KUKA KRL program: EPS_2_25990_SANMH03_A_20260122125456.src

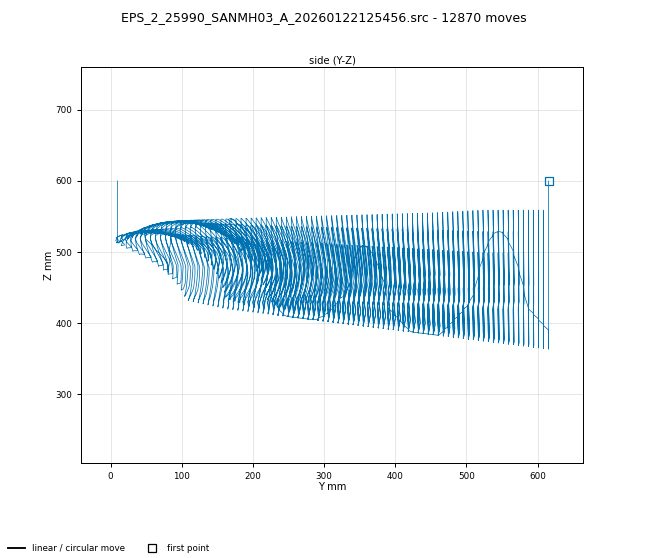
[picture p0: tool path of EPS_2_25990_SANMH03_A_20260122125456.src, 12870 of 12872 moves have a stored position in this frame; points joined in program order, loops and branches not executed]
&ACCESS RVP
&REL 4
&COMMENT QRS 19112012
&PARAM EDITMASK = *
DEF PART()
EXT BAS (BAS_COMMAND :IN,REAL :IN )
INT I
BAS (#INITMOV,0 )

;KUKA QRS Post kuka4.cps  Date:22-06-2017 !

File_ID=3006

QRS_PRE_INIT()

;Init var - Until changes are made in qrs_pre_init
Outlet_Square_prg=0
Inlet_1_Square_prg=0
Inlet_2_Square_prg=0
Inlet_3_Square_prg=0
Inlet_4_Square_prg=0
Inlet_5_Square_prg=0

Outlet_1={X 0.000, Y 520.860, Z 458.500, B 0.000, E1 0.000 }
Inlet_1={X 0.000, Y 523.030, Z 428.500, B 0.000, E1 121.000 }
Inlet_2={X 0.000, Y 529.760, Z 424.000, B 0.000, E1 213.000 }
Outlet_1_type=201
Inlet_1_type=201
Inlet_2_type=150
;QRS#1=Sidecore dimensions
;QRS#2=200-8" PVC SDR 35
;QRS#3=200-8" PVC SDR 35
;QRS#4=150-6" PVC SDR 28
;QRS#5=
;QRS#6=
;QRS#7=
;QRS#8=
;QRS#9=12-08 PSX
;QRS#10=12-08 PSX
;QRS#11=10-06 PSX
;QRS#12=
;QRS#13=
;QRS#14=
;QRS#15=
;QRS#16=1220x127x838 2,75'
;QRS#17=EPS Height
;QRS#18=559
;QRS#19=*
;QRS#20= UPDATED VERSION 22-06-2017
;QRS#21=*
Outlet_Square=0100
Inlet_1_Square=0100
Inlet_2_Square=070
Inlet_3_Square=0
Inlet_4_Square=0
Inlet_5_Square=0
Mill_Square=1
Outlet_Square_Prg=204
Inlet_1_Square_prg=204
Inlet_2_Square_prg=203

QRS_INIT()

$ADVANCE=5

; T1
PTP {E1 173.659,E2 173.659}
PTP {X 0,Y 615.494,A -85,B 0,C 180,E1 173.659,E2 173.659,E3 0,E4 0,E5 0,E6 0}
QRS_SPEED_INIT()
LIN {X 0,Y 615.494,Z 600,A -85,B 0,C 180,E1 173.659,E2 173.659,E3 0,E4 0,E5 0,E6 0} C_VEL
LIN {X 0,Y 615.494,Z 399.527,A -85,B 0,C 180,E1 173.659,E2 173.659} C_VEL
LIN {X 0,Y 615.494,Z 391.592,A -85,B 0,C 180,E1 173.659,E2 173.659} C_VEL
LIN {X 0,Y 615.477,Z 389.645,A -85,B 0,C 180,E1 173.431,E2 173.431} C_VEL
LIN {X 0,Y 615.481,Z 396.286,A -85,B 0,C 180,E1 170.801,E2 170.801} C_VEL
LIN {X 0,Y 615.485,Z 403.113,A -85,B 0,C 180,E1 168.139,E2 168.139} C_VEL
LIN {X 0,Y 615.478,Z 410.131,A -85,B 0,C 180,E1 165.451,E2 165.451} C_VEL
LIN {X 0,Y 615.485,Z 417.333,A -85,B 0,C 180,E1 162.73,E2 162.73} C_VEL
LIN {X 0,Y 615.493,Z 423.081,A -85,B 0,C 180,E1 160.576,E2 160.576} C_VEL
LIN {X 0,Y 615.483,Z 435.817,A -85,B 0,C 180,E1 160.315,E2 160.315} C_VEL
LIN {X 0,Y 615.464,Z 449.029,A -85,B 0,C 180,E1 159.902,E2 159.902} C_VEL
LIN {X 0,Y 615.483,Z 461.622,A -85,B 0,C 180,E1 159.358,E2 159.358} C_VEL
LIN {X 0,Y 615.489,Z 472.571,A -85,B 0,C 180,E1 158.744,E2 158.744} C_VEL
LIN {X 0,Y 615.498,Z 483.738,A -85,B 0,C 180,E1 157.952,E2 157.952} C_VEL
LIN {X 0,Y 615.498,Z 492.862,A -85,B 0,C 180,E1 157.156,E2 157.156} C_VEL
LIN {X 0,Y 615.497,Z 501.581,A -85,B 0,C 180,E1 156.217,E2 156.217} C_VEL
LIN {X 0,Y 615.498,Z 509.269,A -85,B 0,C 180,E1 155.189,E2 155.189} C_VEL
LIN {X 0,Y 615.498,Z 514.717,A -85,B 0,C 180,E1 154.285,E2 154.285} C_VEL
LIN {X 0,Y 615.499,Z 519.658,A -85,B 0,C 180,E1 153.256,E2 153.256} C_VEL
LIN {X 0,Y 615.496,Z 523.851,A -85,B 0,C 180,E1 152.086,E2 152.086} C_VEL
LIN {X 0,Y 615.495,Z 525.744,A -85,B 0,C 180,E1 151.343,E2 151.343} C_VEL
LIN {X 0,Y 615.499,Z 527.649,A -85,B 0,C 180,E1 150.204,E2 150.204} C_VEL
LIN {X 0,Y 615.492,Z 528.385,A -85,B 0,C 180,E1 148.914,E2 148.914} C_VEL
LIN {X 0,Y 615.497,Z 527.605,A -85,B 0,C 180,E1 147.668,E2 147.668} C_VEL
LIN {X 0,Y 615.497,Z 525.522,A -85,B 0,C 180,E1 146.465,E2 146.465} C_VEL
LIN {X 0,Y 615.499,Z 521.736,A -85,B 0,C 180,E1 145.186,E2 145.186} C_VEL
LIN {X 0,Y 615.497,Z 517.474,A -85,B 0,C 180,E1 144.166,E2 144.166} C_VEL
LIN {X 0,Y 615.497,Z 511.462,A -85,B 0,C 180,E1 143.063,E2 143.063} C_VEL
LIN {X 0,Y 615.494,Z 503.996,A -85,B 0,C 180,E1 141.988,E2 141.988} C_VEL
LIN {X 0,Y 615.498,Z 496.26,A -85,B 0,C 180,E1 141.097,E2 141.097} C_VEL
LIN {X 0,Y 615.495,Z 487.302,A -85,B 0,C 180,E1 140.251,E2 140.251} C_VEL
LIN {X 0,Y 615.498,Z 477.935,A -85,B 0,C 180,E1 139.524,E2 139.524} C_VEL
LIN {X 0,Y 615.427,Z 466.634,A -85,B 0,C 180,E1 138.814,E2 138.814} C_VEL
LIN {X 0,Y 615.417,Z 454.465,A -85,B 0,C 180,E1 138.223,E2 138.223} C_VEL
LIN {X 0,Y 615.453,Z 442.53,A -85,B 0,C 180,E1 137.786,E2 137.786} C_VEL
LIN {X 0,Y 615.497,Z 429.773,A -85,B 0,C 180,E1 137.457,E2 137.457} C_VEL
LIN {X 0,Y 615.475,Z 423.066,A -85,B 0,C 180,E1 137.327,E2 137.327} C_VEL
LIN {X 0,Y 615.428,Z 416.675,A -85,B 0,C 180,E1 134.926,E2 134.926} C_VEL
LIN {X 0,Y 615.42,Z 409.882,A -85,B 0,C 180,E1 132.359,E2 132.359} C_VEL
LIN {X 0,Y 615.486,Z 403.062,A -85,B 0,C 180,E1 129.751,E2 129.751} C_VEL
LIN {X 0,Y 615.43,Z 395.839,A -85,B 0,C 180,E1 126.93,E2 126.93} C_VEL
LIN {X 0,Y 615.426,Z 390.192,A -85,B 0,C 180,E1 124.693,E2 124.693} C_VEL
LIN {X 0,Y 615.446,Z 384.318,A -85,B 0,C 180,E1 122.325,E2 122.325} C_VEL
LIN {X 0,Y 615.466,Z 377.257,A -85,B 0,C 180,E1 119.408,E2 119.408} C_VEL
LIN {X 0,Y 615.473,Z 371.567,A -85,B 0,C 180,E1 117.043,E2 117.043} C_VEL
LIN {X 0,Y 615.487,Z 364.488,A -85,B 0,C 180,E1 114.273,E2 114.273} C_VEL
LIN {X 0,Y 615.495,Z 363.693,A -85,B 0,C 180,E1 113.897,E2 113.897} C_VEL
LIN {X 0,Y 615.487,Z 363.694,A -85,B 0,C 180,E1 111.433,E2 111.433} C_VEL
LIN {X 0,Y 615.445,Z 363.7,A -85,B 0,C 180,E1 108.594,E2 108.594} C_VEL
LIN {X 0,Y 615.49,Z 363.691,A -85,B 0,C 180,E1 105.906,E2 105.906} C_VEL
LIN {X 0,Y 615.492,Z 363.7,A -85,B 0,C 180,E1 103.202,E2 103.202} C_VEL
LIN {X 0,Y 615.458,Z 363.7,A -85,B 0,C 180,E1 100.529,E2 100.529} C_VEL
LIN {X 0,Y 615.489,Z 363.69,A -85,B 0,C 180,E1 97.877,E2 97.877} C_VEL
LIN {X 0,Y 615.476,Z 363.7,A -85,B 0,C 180,E1 95.243,E2 95.243} C_VEL
LIN {X 0,Y 615.461,Z 363.701,A -85,B 0,C 180,E1 92.619,E2 92.619} C_VEL
LIN {X 0,Y 615.485,Z 363.692,A -85,B 0,C 180,E1 89.674,E2 89.674} C_VEL
LIN {X 0,Y 615.49,Z 363.848,A -85,B 0,C 180,E1 89.347,E2 89.347} C_VEL
LIN {X 0,Y 615.489,Z 369.621,A -85,B 0,C 180,E1 86.729,E2 86.729} C_VEL
LIN {X 0,Y 615.496,Z 375.508,A -85,B 0,C 180,E1 84.103,E2 84.103} C_VEL
LIN {X 0,Y 615.474,Z 381.581,A -85,B 0,C 180,E1 81.465,E2 81.465} C_VEL
LIN {X 0,Y 615.479,Z 387.798,A -85,B 0,C 180,E1 78.809,E2 78.809} C_VEL
LIN {X 0,Y 615.494,Z 394.357,A -85,B 0,C 180,E1 76.064,E2 76.064} C_VEL
LIN {X 0,Y 615.485,Z 400.781,A -85,B 0,C 180,E1 73.415,E2 73.415} C_VEL
LIN {X 0,Y 615.459,Z 407.558,A -85,B 0,C 180,E1 70.663,E2 70.663} C_VEL
LIN {X 0,Y 615.493,Z 414.508,A -85,B 0,C 180,E1 67.866,E2 67.866} C_VEL
LIN {X 0,Y 615.496,Z 419.067,A -85,B 0,C 180,E1 66.103,E2 66.103} C_VEL
LIN {X 0,Y 615.478,Z 430.982,A -85,B 0,C 180,E1 65.794,E2 65.794} C_VEL
LIN {X 0,Y 615.446,Z 439.974,A -85,B 0,C 180,E1 65.459,E2 65.459} C_VEL
LIN {X 0,Y 615.436,Z 449.191,A -85,B 0,C 180,E1 65.008,E2 65.008} C_VEL
LIN {X 0,Y 615.47,Z 457.359,A -85,B 0,C 180,E1 64.504,E2 64.504} C_VEL
LIN {X 0,Y 615.499,Z 465.031,A -85,B 0,C 180,E1 63.923,E2 63.923} C_VEL
LIN {X 0,Y 615.496,Z 473.758,A -85,B 0,C 180,E1 63.104,E2 63.104} C_VEL
LIN {X 0,Y 615.499,Z 480.59,A -85,B 0,C 180,E1 62.273,E2 62.273} C_VEL
LIN {X 0,Y 615.497,Z 485.434,A -85,B 0,C 180,E1 61.548,E2 61.548} C_VEL
LIN {X 0,Y 615.492,Z 488.696,A -85,B 0,C 180,E1 60.971,E2 60.971} C_VEL
LIN {X 0,Y 615.498,Z 492.162,A -85,B 0,C 180,E1 60.203,E2 60.203} C_VEL
LIN {X 0,Y 615.496,Z 494.722,A -85,B 0,C 180,E1 59.464,E2 59.464} C_VEL
LIN {X 0,Y 615.495,Z 497.253,A -85,B 0,C 180,E1 58.318,E2 58.318} C_VEL
LIN {X 0,Y 615.496,Z 498.133,A -85,B 0,C 180,E1 57.546,E2 57.546} C_VEL
LIN {X 0,Y 615.492,Z 498.18,A -85,B 0,C 180,E1 56.465,E2 56.465} C_VEL
LIN {X 0,Y 615.492,Z 496.809,A -85,B 0,C 180,E1 55.298,E2 55.298} C_VEL
LIN {X 0,Y 615.491,Z 493.761,A -85,B 0,C 180,E1 54.166,E2 54.166} C_VEL
LIN {X 0,Y 615.497,Z 490.45,A -85,B 0,C 180,E1 53.321,E2 53.321} C_VEL
LIN {X 0,Y 615.493,Z 486.628,A -85,B 0,C 180,E1 52.568,E2 52.568} C_VEL
LIN {X 0,Y 615.496,Z 482.71,A -85,B 0,C 180,E1 51.935,E2 51.935} C_VEL
LIN {X 0,Y 615.498,Z 476.29,A -85,B 0,C 180,E1 51.099,E2 51.099} C_VEL
LIN {X 0,Y 615.499,Z 469.919,A -85,B 0,C 180,E1 50.425,E2 50.425} C_VEL
LIN {X 0,Y 615.474,Z 460.924,A -85,B 0,C 180,E1 49.652,E2 49.652} C_VEL
LIN {X 0,Y 615.455,Z 451.474,A -85,B 0,C 180,E1 49.03,E2 49.03} C_VEL
LIN {X 0,Y 615.487,Z 442.766,A -85,B 0,C 180,E1 48.577,E2 48.577} C_VEL
LIN {X 0,Y 615.494,Z 434.152,A -85,B 0,C 180,E1 48.225,E2 48.225} C_VEL
LIN {X 0,Y 615.491,Z 425.461,A -85,B 0,C 180,E1 47.958,E2 47.958} C_VEL
LIN {X 0,Y 615.48,Z 418.875,A -85,B 0,C 180,E1 47.784,E2 47.784} C_VEL
LIN {X 0,Y 615.455,Z 411.74,A -85,B 0,C 180,E1 44.932,E2 44.932} C_VEL
LIN {X 0,Y 615.469,Z 404.683,A -85,B 0,C 180,E1 42.082,E2 42.082} C_VEL
LIN {X 0,Y 615.426,Z 398.996,A -85,B 0,C 180,E1 39.755,E2 39.755} C_VEL
LIN {X 0,Y 615.43,Z 394.77,A -85,B 0,C 180,E1 38.009,E2 38.009} C_VEL
LIN {X 0,Y 615.423,Z 389.043,A -85,B 0,C 180,E1 35.62,E2 35.62} C_VEL
LIN {X 0,Y 615.455,Z 383.422,A -85,B 0,C 180,E1 33.238,E2 33.238} C_VEL
LIN {X 0,Y 615.491,Z 378.051,A -85,B 0,C 180,E1 30.919,E2 30.919} C_VEL
LIN {X 0,Y 615.473,Z 372.464,A -85,B 0,C 180,E1 28.453,E2 28.453} C_VEL
LIN {X 0,Y 615.494,Z 366.375,A -85,B 0,C 180,E1 25.715,E2 25.715} C_VEL
LIN {X 0,Y 615.473,Z 363.7,A -85,B 0,C 180,E1 24.452,E2 24.452} C_VEL
LIN {X 0,Y 615.496,Z 363.699,A -85,B 0,C 180,E1 22.136,E2 22.136} C_VEL
LIN {X 0,Y 615.489,Z 363.701,A -85,B 0,C 180,E1 19.338,E2 19.338} C_VEL
LIN {X 0,Y 615.485,Z 363.7,A -85,B 0,C 180,E1 16.586,E2 16.586} C_VEL
LIN {X 0,Y 615.483,Z 363.699,A -85,B 0,C 180,E1 13.874,E2 13.874} C_VEL
LIN {X 0,Y 615.489,Z 363.694,A -85,B 0,C 180,E1 10.904,E2 10.904} C_VEL
LIN {X 0,Y 615.482,Z 363.7,A -85,B 0,C 180,E1 8.536,E2 8.536} C_VEL
LIN {X 0,Y 615.487,Z 363.7,A -85,B 0,C 180,E1 5.898,E2 5.898} C_VEL
LIN {X 0,Y 615.492,Z 363.7,A -85,B 0,C 180,E1 3.273,E2 3.273} C_VEL
LIN {X 0,Y 615.489,Z 363.701,A -85,B 0,C 180,E1 0.654,E2 0.654} C_VEL
LIN {X 0,Y 615.498,Z 363.7,A -85,B 0,C 180,E1 -1.963,E2 -1.963} C_VEL
LIN {X 0,Y 615.489,Z 363.701,A -85,B 0,C 180,E1 -4.585,E2 -4.585} C_VEL
LIN {X 0,Y 615.492,Z 363.699,A -85,B 0,C 180,E1 -7.216,E2 -7.216} C_VEL
LIN {X 0,Y 615.487,Z 363.7,A -85,B 0,C 180,E1 -9.862,E2 -9.862} C_VEL
LIN {X 0,Y 615.485,Z 363.7,A -85,B 0,C 180,E1 -12.53,E2 -12.53} C_VEL
LIN {X 0,Y 615.491,Z 363.699,A -85,B 0,C 180,E1 -15.226,E2 -15.226} C_VEL
LIN {X 0,Y 615.49,Z 363.701,A -85,B 0,C 180,E1 -17.957,E2 -17.957} C_VEL
LIN {X 0,Y 615.492,Z 363.701,A -85,B 0,C 180,E1 -20.731,E2 -20.731} C_VEL
LIN {X 0,Y 615.478,Z 363.7,A -85,B 0,C 180,E1 -23.557,E2 -23.557} C_VEL
LIN {X 0,Y 615.488,Z 363.695,A -85,B 0,C 180,E1 -26.444,E2 -26.444} C_VEL
LIN {X 0,Y 615.459,Z 363.7,A -85,B 0,C 180,E1 -29.408,E2 -29.408} C_VEL
LIN {X 0,Y 615.472,Z 363.7,A -85,B 0,C 180,E1 -31.687,E2 -31.687} C_VEL
LIN {X 0,Y 615.492,Z 363.692,A -85,B 0,C 180,E1 -34.706,E2 -34.706} C_VEL
LIN {X 0,Y 615.457,Z 363.701,A -85,B 0,C 180,E1 -37.245,E2 -37.245} C_VEL
LIN {X 0,Y 615.473,Z 363.699,A -85,B 0,C 180,E1 -39.752,E2 -39.752} C_VEL
LIN {X 0,Y 615.495,Z 363.695,A -85,B 0,C 180,E1 -42.353,E2 -42.353} C_VEL
LIN {X 0,Y 615.468,Z 363.7,A -85,B 0,C 180,E1 -45.071,E2 -45.071} C_VEL
LIN {X 0,Y 615.474,Z 363.697,A -85,B 0,C 180,E1 -47.922,E2 -47.922} C_VEL
LIN {X 0,Y 615.477,Z 363.697,A -85,B 0,C 180,E1 -50.94,E2 -50.94} C_VEL
LIN {X 0,Y 615.46,Z 363.7,A -85,B 0,C 180,E1 -53.576,E2 -53.576} C_VEL
LIN {X 0,Y 615.492,Z 363.695,A -85,B 0,C 180,E1 -56.466,E2 -56.466} C_VEL
LIN {X 0,Y 615.477,Z 363.698,A -85,B 0,C 180,E1 -59.082,E2 -59.082} C_VEL
LIN {X 0,Y 615.49,Z 363.711,A -85,B 0,C 180,E1 -60.303,E2 -60.303} C_VEL
LIN {X 0,Y 615.449,Z 375.744,A -85,B 0,C 180,E1 -62.963,E2 -62.963} C_VEL
LIN {X 0,Y 615.43,Z 385.189,A -85,B 0,C 180,E1 -65.008,E2 -65.008} C_VEL
LIN {X 0,Y 615.446,Z 396.451,A -85,B 0,C 180,E1 -67.408,E2 -67.408} C_VEL
LIN {X 0,Y 615.494,Z 408.677,A -85,B 0,C 180,E1 -69.97,E2 -69.97} C_VEL
LIN {X 0,Y 615.472,Z 422.09,A -85,B 0,C 180,E1 -72.731,E2 -72.731} C_VEL
LIN {X 0,Y 615.475,Z 435.487,A -85,B 0,C 180,E1 -75.453,E2 -75.453} C_VEL
LIN {X 0,Y 615.488,Z 448.873,A -85,B 0,C 180,E1 -78.141,E2 -78.141} C_VEL
LIN {X 0,Y 615.494,Z 449.811,A -85,B 0,C 180,E1 -78.329,E2 -78.329} C_VEL
LIN {X 0,Y 615.498,Z 464.14,A -85,B 0,C 180,E1 -78.6,E2 -78.6} C_VEL
LIN {X 0,Y 615.463,Z 476.758,A -85,B 0,C 180,E1 -78.969,E2 -78.969} C_VEL
LIN {X 0,Y 615.451,Z 489.065,A -85,B 0,C 180,E1 -79.474,E2 -79.474} C_VEL
LIN {X 0,Y 615.486,Z 500.011,A -85,B 0,C 180,E1 -80.057,E2 -80.057} C_VEL
LIN {X 0,Y 615.499,Z 511.19,A -85,B 0,C 180,E1 -80.803,E2 -80.803} C_VEL
LIN {X 0,Y 615.498,Z 521.063,A -85,B 0,C 180,E1 -81.631,E2 -81.631} C_VEL
LIN {X 0,Y 615.498,Z 530.62,A -85,B 0,C 180,E1 -82.621,E2 -82.621} C_VEL
LIN {X 0,Y 615.496,Z 538.214,A -85,B 0,C 180,E1 -83.61,E2 -83.61} C_VEL
LIN {X 0,Y 615.498,Z 545.213,A -85,B 0,C 180,E1 -84.76,E2 -84.76} C_VEL
LIN {X 0,Y 615.494,Z 549.858,A -85,B 0,C 180,E1 -85.745,E2 -85.745} C_VEL
LIN {X 0,Y 615.494,Z 553.404,A -85,B 0,C 180,E1 -86.729,E2 -86.729} C_VEL
LIN {X 0,Y 615.497,Z 555.237,A -85,B 0,C 180,E1 -87.384,E2 -87.384} C_VEL
LIN {X 0,Y 615.499,Z 556.61,A -85,B 0,C 180,E1 -88.038,E2 -88.038} C_VEL
LIN {X 0,Y 615.496,Z 558.175,A -85,B 0,C 180,E1 -89.347,E2 -89.347} C_VEL
LIN {X 0,Y 615.494,Z 558.389,A -85,B 0,C 180,E1 -90.001,E2 -90.001} C_VEL
LIN {X 0,Y 615.495,Z 557.578,A -85,B 0,C 180,E1 -91.31,E2 -91.31} C_VEL
LIN {X 0,Y 615.499,Z 556.605,A -85,B 0,C 180,E1 -91.964,E2 -91.964} C_VEL
LIN {X 0,Y 615.497,Z 555.229,A -85,B 0,C 180,E1 -92.619,E2 -92.619} C_VEL
LIN {X 0,Y 615.496,Z 552.345,A -85,B 0,C 180,E1 -93.602,E2 -93.602} C_VEL
LIN {X 0,Y 615.498,Z 548.436,A -85,B 0,C 180,E1 -94.586,E2 -94.586} C_VEL
LIN {X 0,Y 615.499,Z 543.397,A -85,B 0,C 180,E1 -95.571,E2 -95.571} C_VEL
LIN {X 0,Y 615.497,Z 536.87,A -85,B 0,C 180,E1 -96.583,E2 -96.583} C_VEL
LIN {X 0,Y 615.497,Z 529.122,A -85,B 0,C 180,E1 -97.547,E2 -97.547} C_VEL
LIN {X 0,Y 615.498,Z 521.031,A -85,B 0,C 180,E1 -98.372,E2 -98.372} C_VEL
LIN {X 0,Y 615.499,Z 511.151,A -85,B 0,C 180,E1 -99.2,E2 -99.2} C_VEL
LIN {X 0,Y 615.488,Z 499.961,A -85,B 0,C 180,E1 -99.946,E2 -99.946} C_VEL
LIN {X 0,Y 615.452,Z 489.003,A -85,B 0,C 180,E1 -100.529,E2 -100.529} C_VEL
LIN {X 0,Y 615.464,Z 476.705,A -85,B 0,C 180,E1 -101.033,E2 -101.033} C_VEL
LIN {X 0,Y 615.498,Z 464.01,A -85,B 0,C 180,E1 -101.403,E2 -101.403} C_VEL
LIN {X 0,Y 615.494,Z 449.797,A -85,B 0,C 180,E1 -101.674,E2 -101.674} C_VEL
LIN {X 0,Y 615.475,Z 437.007,A -85,B 0,C 180,E1 -104.242,E2 -104.242} C_VEL
LIN {X 0,Y 615.481,Z 423.747,A -85,B 0,C 180,E1 -106.93,E2 -106.93} C_VEL
LIN {X 0,Y 615.483,Z 410.342,A -85,B 0,C 180,E1 -109.686,E2 -109.686} C_VEL
LIN {X 0,Y 615.467,Z 397.638,A -85,B 0,C 180,E1 -112.341,E2 -112.341} C_VEL
LIN {X 0,Y 615.427,Z 386.854,A -85,B 0,C 180,E1 -114.635,E2 -114.635} C_VEL
LIN {X 0,Y 615.449,Z 375.744,A -85,B 0,C 180,E1 -117.037,E2 -117.037} C_VEL
LIN {X 0,Y 615.485,Z 363.69,A -85,B 0,C 180,E1 -119.721,E2 -119.721} C_VEL
LIN {X 0,Y 615.472,Z 363.695,A -85,B 0,C 180,E1 -122.459,E2 -122.459} C_VEL
LIN {X 0,Y 615.486,Z 363.697,A -85,B 0,C 180,E1 -124.816,E2 -124.816} C_VEL
LIN {X 0,Y 615.474,Z 363.689,A -85,B 0,C 180,E1 -127.244,E2 -127.244} C_VEL
LIN {X 0,Y 615.488,Z 363.7,A -85,B 0,C 180,E1 -130.089,E2 -130.089} C_VEL
LIN {X 0,Y 615.439,Z 363.699,A -85,B 0,C 180,E1 -132.358,E2 -132.358} C_VEL
LIN {X 0,Y 615.455,Z 363.701,A -85,B 0,C 180,E1 -135.072,E2 -135.072} C_VEL
LIN {X 0,Y 615.456,Z 363.693,A -85,B 0,C 180,E1 -137.924,E2 -137.924} C_VEL
LIN {X 0,Y 615.463,Z 363.695,A -85,B 0,C 180,E1 -140.248,E2 -140.248} C_VEL
LIN {X 0,Y 615.483,Z 363.69,A -85,B 0,C 180,E1 -143.064,E2 -143.064} C_VEL
LIN {X 0,Y 615.488,Z 363.686,A -85,B 0,C 180,E1 -145.3,E2 -145.3} C_VEL
LIN {X 0,Y 615.493,Z 363.694,A -85,B 0,C 180,E1 -147.669,E2 -147.669} C_VEL
LIN {X 0,Y 615.448,Z 363.698,A -85,B 0,C 180,E1 -150.212,E2 -150.212} C_VEL
LIN {X 0,Y 615.435,Z 363.7,A -85,B 0,C 180,E1 -152.082,E2 -152.082} C_VEL
LIN {X 0,Y 615.431,Z 363.7,A -85,B 0,C 180,E1 -154.443,E2 -154.443} C_VEL
LIN {X 0,Y 615.497,Z 363.692,A -85,B 0,C 180,E1 -157.156,E2 -157.156} C_VEL
LIN {X 0,Y 615.461,Z 363.695,A -85,B 0,C 180,E1 -159.966,E2 -159.966} C_VEL
LIN {X 0,Y 615.48,Z 363.691,A -85,B 0,C 180,E1 -162.729,E2 -162.729} C_VEL
LIN {X 0,Y 615.49,Z 363.691,A -85,B 0,C 180,E1 -165.451,E2 -165.451} C_VEL
LIN {X 0,Y 615.454,Z 363.697,A -85,B 0,C 180,E1 -168.138,E2 -168.138} C_VEL
LIN {X 0,Y 615.462,Z 363.697,A -85,B 0,C 180,E1 -170.801,E2 -170.801} C_VEL
LIN {X 0,Y 615.453,Z 363.698,A -85,B 0,C 180,E1 -173.45,E2 -173.45} C_VEL
LIN {X 0,Y 615.449,Z 363.698,A -85,B 0,C 180,E1 -176.071,E2 -176.071} C_VEL
LIN {X 0,Y 615.476,Z 363.974,A -85,B 0,C 180,E1 -176.399,E2 -176.399} C_VEL
LIN {X 0,Y 615.489,Z 370.297,A -85,B 0,C 180,E1 -178.691,E2 -178.691} C_VEL
LIN {X 0,Y 615.482,Z 375.236,A -85,B 0,C 180,E1 -180.654,E2 -180.654} C_VEL
LIN {X 0,Y 615.48,Z 381.527,A -85,B 0,C 180,E1 -183.273,E2 -183.273} C_VEL
LIN {X 0,Y 615.497,Z 387.971,A -85,B 0,C 180,E1 -185.898,E2 -185.898} C_VEL
LIN {X 0,Y 615.477,Z 389.645,A -85,B 0,C 180,E1 -186.569,E2 -186.569} C_VEL
LIN {X 0,Y 614.8,Z 391.13,A -85,B 0,C 180,E1 -187.099,E2 -187.099} C_VEL
LIN {X 0,Y 611.944,Z 393.686,A -85,B 0,C 180,E1 -187.953,E2 -187.953} C_VEL
LIN {X 0,Y 609.543,Z 395.676,A -85,B 0,C 180,E1 -188.64,E2 -188.64} C_VEL
LIN {X 0,Y 608.513,Z 397.105,A -85,B 0,C 180,E1 -189.172,E2 -189.172} C_VEL
LIN {X 0,Y 608.431,Z 397.568,A -85,B 0,C 180,E1 -189.353,E2 -189.353} C_VEL
LIN {X 0,Y 608.425,Z 404.335,A -85,B 0,C 180,E1 -192,E2 -192} C_VEL
LIN {X 0,Y 608.436,Z 411.401,A -85,B 0,C 180,E1 -194.721,E2 -194.721} C_VEL
LIN {X 0,Y 608.429,Z 418.66,A -85,B 0,C 180,E1 -197.477,E2 -197.477} C_VEL
LIN {X 0,Y 608.432,Z 423.472,A -85,B 0,C 180,E1 -199.286,E2 -199.286} C_VEL
LIN {X 0,Y 608.523,Z 438.048,A -85,B 0,C 180,E1 -199.612,E2 -199.612} C_VEL
LIN {X 0,Y 608.503,Z 451.304,A -85,B 0,C 180,E1 -200.052,E2 -200.052} C_VEL
LIN {X 0,Y 608.513,Z 463.064,A -85,B 0,C 180,E1 -200.587,E2 -200.587} C_VEL
LIN {X 0,Y 608.486,Z 474.347,A -85,B 0,C 180,E1 -201.246,E2 -201.246} C_VEL
LIN {X 0,Y 608.497,Z 485.298,A -85,B 0,C 180,E1 -202.047,E2 -202.047} C_VEL
LIN {X 0,Y 608.475,Z 494.924,A -85,B 0,C 180,E1 -202.925,E2 -202.925} C_VEL
LIN {X 0,Y 608.445,Z 503.147,A -85,B 0,C 180,E1 -203.846,E2 -203.846} C_VEL
LIN {X 0,Y 608.456,Z 510.996,A -85,B 0,C 180,E1 -204.935,E2 -204.935} C_VEL
LIN {X 0,Y 608.437,Z 517.174,A -85,B 0,C 180,E1 -206.036,E2 -206.036} C_VEL
LIN {X 0,Y 608.435,Z 522.153,A -85,B 0,C 180,E1 -207.199,E2 -207.199} C_VEL
LIN {X 0,Y 608.441,Z 525.464,A -85,B 0,C 180,E1 -208.267,E2 -208.267} C_VEL
LIN {X 0,Y 608.42,Z 527.14,A -85,B 0,C 180,E1 -209.022,E2 -209.022} C_VEL
LIN {X 0,Y 608.423,Z 528.469,A -85,B 0,C 180,E1 -209.964,E2 -209.964} C_VEL
LIN {X 0,Y 608.439,Z 528.887,A -85,B 0,C 180,E1 -210.546,E2 -210.546} C_VEL
LIN {X 0,Y 608.422,Z 528.942,A -85,B 0,C 180,E1 -211.319,E2 -211.319} C_VEL
LIN {X 0,Y 608.422,Z 528.01,A -85,B 0,C 180,E1 -212.516,E2 -212.516} C_VEL
LIN {X 0,Y 608.424,Z 525.719,A -85,B 0,C 180,E1 -213.727,E2 -213.727} C_VEL
LIN {X 0,Y 608.429,Z 522.112,A -85,B 0,C 180,E1 -214.902,E2 -214.902} C_VEL
LIN {X 0,Y 608.456,Z 516.993,A -85,B 0,C 180,E1 -216.091,E2 -216.091} C_VEL
LIN {X 0,Y 608.439,Z 511.004,A -85,B 0,C 180,E1 -217.154,E2 -217.154} C_VEL
LIN {X 0,Y 608.458,Z 503.196,A -85,B 0,C 180,E1 -218.238,E2 -218.238} C_VEL
LIN {X 0,Y 608.483,Z 495.025,A -85,B 0,C 180,E1 -219.155,E2 -219.155} C_VEL
LIN {X 0,Y 608.489,Z 486.121,A -85,B 0,C 180,E1 -219.976,E2 -219.976} C_VEL
LIN {X 0,Y 608.482,Z 476,A -85,B 0,C 180,E1 -220.736,E2 -220.736} C_VEL
LIN {X 0,Y 608.428,Z 464.384,A -85,B 0,C 180,E1 -221.434,E2 -221.434} C_VEL
LIN {X 0,Y 608.456,Z 452.111,A -85,B 0,C 180,E1 -222.007,E2 -222.007} C_VEL
LIN {X 0,Y 608.513,Z 439.113,A -85,B 0,C 180,E1 -222.449,E2 -222.449} C_VEL
LIN {X 0,Y 608.539,Z 425.565,A -85,B 0,C 180,E1 -222.757,E2 -222.757} C_VEL
LIN {X 0,Y 608.414,Z 423.473,A -85,B 0,C 180,E1 -222.804,E2 -222.804} C_VEL
LIN {X 0,Y 608.362,Z 417.125,A -85,B 0,C 180,E1 -225.195,E2 -225.195} C_VEL
LIN {X 0,Y 608.383,Z 409.935,A -85,B 0,C 180,E1 -227.931,E2 -227.931} C_VEL
LIN {X 0,Y 608.418,Z 402.744,A -85,B 0,C 180,E1 -230.708,E2 -230.708} C_VEL
LIN {X 0,Y 608.395,Z 395.662,A -85,B 0,C 180,E1 -233.493,E2 -233.493} C_VEL
LIN {X 0,Y 608.445,Z 388.591,A -85,B 0,C 180,E1 -236.327,E2 -236.327} C_VEL
LIN {X 0,Y 608.434,Z 382.719,A -85,B 0,C 180,E1 -238.734,E2 -238.734} C_VEL
LIN {X 0,Y 608.41,Z 377.366,A -85,B 0,C 180,E1 -240.976,E2 -240.976} C_VEL
LIN {X 0,Y 608.429,Z 371.805,A -85,B 0,C 180,E1 -243.224,E2 -243.224} C_VEL
LIN {X 0,Y 608.46,Z 365.141,A -85,B 0,C 180,E1 -245.851,E2 -245.851} C_VEL
LIN {X 0,Y 608.48,Z 364.69,A -85,B 0,C 180,E1 -246.155,E2 -246.155} C_VEL
LIN {X 0,Y 608.468,Z 364.69,A -85,B 0,C 180,E1 -248.307,E2 -248.307} C_VEL
LIN {X 0,Y 608.437,Z 364.693,A -85,B 0,C 180,E1 -251.129,E2 -251.129} C_VEL
LIN {X 0,Y 608.464,Z 364.693,A -85,B 0,C 180,E1 -253.905,E2 -253.905} C_VEL
LIN {X 0,Y 608.47,Z 364.695,A -85,B 0,C 180,E1 -256.643,E2 -256.643} C_VEL
LIN {X 0,Y 608.433,Z 364.695,A -85,B 0,C 180,E1 -259.348,E2 -259.348} C_VEL
LIN {X 0,Y 608.481,Z 364.688,A -85,B 0,C 180,E1 -262.032,E2 -262.032} C_VEL
LIN {X 0,Y 608.458,Z 364.696,A -85,B 0,C 180,E1 -264.697,E2 -264.697} C_VEL
LIN {X 0,Y 608.453,Z 364.694,A -85,B 0,C 180,E1 -267.35,E2 -267.35} C_VEL
LIN {X 0,Y 608.48,Z 364.688,A -85,B 0,C 180,E1 -269.999,E2 -269.999} C_VEL
LIN {X 0,Y 608.484,Z 364.881,A -85,B 0,C 180,E1 -270.66,E2 -270.66} C_VEL
LIN {X 0,Y 608.453,Z 370.695,A -85,B 0,C 180,E1 -273.309,E2 -273.309} C_VEL
LIN {X 0,Y 608.466,Z 376.611,A -85,B 0,C 180,E1 -275.965,E2 -275.965} C_VEL
LIN {X 0,Y 608.447,Z 382.709,A -85,B 0,C 180,E1 -278.634,E2 -278.634} C_VEL
LIN {X 0,Y 608.442,Z 388.979,A -85,B 0,C 180,E1 -281.323,E2 -281.323} C_VEL
LIN {X 0,Y 608.446,Z 395.428,A -85,B 0,C 180,E1 -284.036,E2 -284.036} C_VEL
LIN {X 0,Y 608.438,Z 402.064,A -85,B 0,C 180,E1 -286.783,E2 -286.783} C_VEL
LIN {X 0,Y 608.419,Z 407.168,A -85,B 0,C 180,E1 -288.869,E2 -288.869} C_VEL
LIN {X 0,Y 608.401,Z 414.149,A -85,B 0,C 180,E1 -291.692,E2 -291.692} C_VEL
LIN {X 0,Y 608.44,Z 419.345,A -85,B 0,C 180,E1 -293.776,E2 -293.776} C_VEL
LIN {X 0,Y 608.483,Z 431.922,A -85,B 0,C 180,E1 -294.124,E2 -294.124} C_VEL
LIN {X 0,Y 608.442,Z 440.087,A -85,B 0,C 180,E1 -294.434,E2 -294.434} C_VEL
LIN {X 0,Y 608.41,Z 448.545,A -85,B 0,C 180,E1 -294.844,E2 -294.844} C_VEL
LIN {X 0,Y 608.443,Z 457.188,A -85,B 0,C 180,E1 -295.372,E2 -295.372} C_VEL
LIN {X 0,Y 608.481,Z 465.852,A -85,B 0,C 180,E1 -296.032,E2 -296.032} C_VEL
LIN {X 0,Y 608.448,Z 473.694,A -85,B 0,C 180,E1 -296.772,E2 -296.772} C_VEL
LIN {X 0,Y 608.443,Z 481.324,A -85,B 0,C 180,E1 -297.703,E2 -297.703} C_VEL
LIN {X 0,Y 608.445,Z 486.166,A -85,B 0,C 180,E1 -298.438,E2 -298.438} C_VEL
LIN {X 0,Y 608.426,Z 489.398,A -85,B 0,C 180,E1 -299.02,E2 -299.02} C_VEL
LIN {X 0,Y 608.438,Z 493.447,A -85,B 0,C 180,E1 -299.967,E2 -299.967} C_VEL
LIN {X 0,Y 608.441,Z 495.409,A -85,B 0,C 180,E1 -300.544,E2 -300.544} C_VEL
LIN {X 0,Y 608.441,Z 497.293,A -85,B 0,C 180,E1 -301.315,E2 -301.315} C_VEL
LIN {X 0,Y 608.42,Z 498.463,A -85,B 0,C 180,E1 -302.095,E2 -302.095} C_VEL
LIN {X 0,Y 608.415,Z 498.947,A -85,B 0,C 180,E1 -302.879,E2 -302.879} C_VEL
LIN {X 0,Y 608.419,Z 498.704,A -85,B 0,C 180,E1 -303.728,E2 -303.728} C_VEL
LIN {X 0,Y 608.428,Z 496.988,A -85,B 0,C 180,E1 -304.903,E2 -304.903} C_VEL
LIN {X 0,Y 608.426,Z 494.97,A -85,B 0,C 180,E1 -305.682,E2 -305.682} C_VEL
LIN {X 0,Y 608.452,Z 492.006,A -85,B 0,C 180,E1 -306.5,E2 -306.5} C_VEL
LIN {X 0,Y 608.428,Z 487.485,A -85,B 0,C 180,E1 -307.423,E2 -307.423} C_VEL
LIN {X 0,Y 608.455,Z 482.373,A -85,B 0,C 180,E1 -308.239,E2 -308.239} C_VEL
LIN {X 0,Y 608.464,Z 476.379,A -85,B 0,C 180,E1 -309.01,E2 -309.01} C_VEL
LIN {X 0,Y 608.467,Z 469.222,A -85,B 0,C 180,E1 -309.759,E2 -309.759} C_VEL
LIN {X 0,Y 608.449,Z 460.418,A -85,B 0,C 180,E1 -310.496,E2 -310.496} C_VEL
LIN {X 0,Y 608.451,Z 451.779,A -85,B 0,C 180,E1 -311.064,E2 -311.064} C_VEL
LIN {X 0,Y 608.491,Z 442.819,A -85,B 0,C 180,E1 -311.533,E2 -311.533} C_VEL
LIN {X 0,Y 608.499,Z 433.961,A -85,B 0,C 180,E1 -311.894,E2 -311.894} C_VEL
LIN {X 0,Y 608.505,Z 424.89,A -85,B 0,C 180,E1 -312.171,E2 -312.171} C_VEL
LIN {X 0,Y 608.418,Z 419.345,A -85,B 0,C 180,E1 -312.314,E2 -312.314} C_VEL
LIN {X 0,Y 608.41,Z 412.158,A -85,B 0,C 180,E1 -315.2,E2 -315.2} C_VEL
LIN {X 0,Y 608.409,Z 405.418,A -85,B 0,C 180,E1 -317.935,E2 -317.935} C_VEL
LIN {X 0,Y 608.367,Z 399.048,A -85,B 0,C 180,E1 -320.553,E2 -320.553} C_VEL
LIN {X 0,Y 608.406,Z 392.975,A -85,B 0,C 180,E1 -323.082,E2 -323.082} C_VEL
LIN {X 0,Y 608.435,Z 387.191,A -85,B 0,C 180,E1 -325.529,E2 -325.529} C_VEL
LIN {X 0,Y 608.402,Z 381.684,A -85,B 0,C 180,E1 -327.902,E2 -327.902} C_VEL
LIN {X 0,Y 608.429,Z 376.404,A -85,B 0,C 180,E1 -330.219,E2 -330.219} C_VEL
LIN {X 0,Y 608.456,Z 370.666,A -85,B 0,C 180,E1 -332.791,E2 -332.791} C_VEL
LIN {X 0,Y 608.448,Z 364.696,A -85,B 0,C 180,E1 -335.522,E2 -335.522} C_VEL
LIN {X 0,Y 608.455,Z 364.694,A -85,B 0,C 180,E1 -338.308,E2 -338.308} C_VEL
LIN {X 0,Y 608.46,Z 364.692,A -85,B 0,C 180,E1 -341.278,E2 -341.278} C_VEL
LIN {X 0,Y 608.439,Z 364.695,A -85,B 0,C 180,E1 -343.906,E2 -343.906} C_VEL
LIN {X 0,Y 608.457,Z 364.698,A -85,B 0,C 180,E1 -345.976,E2 -345.976} C_VEL
LIN {X 0,Y 608.469,Z 364.696,A -85,B 0,C 180,E1 -348.676,E2 -348.676} C_VEL
LIN {X 0,Y 608.449,Z 364.698,A -85,B 0,C 180,E1 -351.364,E2 -351.364} C_VEL
LIN {X 0,Y 608.481,Z 364.694,A -85,B 0,C 180,E1 -354.034,E2 -354.034} C_VEL
LIN {X 0,Y 608.48,Z 364.694,A -85,B 0,C 180,E1 -356.69,E2 -356.69} C_VEL
LIN {X 0,Y 608.48,Z 364.695,A -85,B 0,C 180,E1 -359.338,E2 -359.338} C_VEL
LIN {X 0,Y 608.467,Z 364.697,A -85,B 0,C 180,E1 -361.986,E2 -361.986} C_VEL
LIN {X 0,Y 608.456,Z 364.698,A -85,B 0,C 180,E1 -364.638,E2 -364.638} C_VEL
LIN {X 0,Y 608.476,Z 364.695,A -85,B 0,C 180,E1 -367.299,E2 -367.299} C_VEL
LIN {X 0,Y 608.455,Z 364.698,A -85,B 0,C 180,E1 -369.978,E2 -369.978} C_VEL
LIN {X 0,Y 608.47,Z 364.696,A -85,B 0,C 180,E1 -372.677,E2 -372.677} C_VEL
LIN {X 0,Y 608.465,Z 364.696,A -85,B 0,C 180,E1 -375.406,E2 -375.406} C_VEL
LIN {X 0,Y 608.45,Z 364.696,A -85,B 0,C 180,E1 -378.172,E2 -378.172} C_VEL
LIN {X 0,Y 608.447,Z 364.695,A -85,B 0,C 180,E1 -380.982,E2 -380.982} C_VEL
LIN {X 0,Y 608.449,Z 364.696,A -85,B 0,C 180,E1 -383.124,E2 -383.124} C_VEL
LIN {X 0,Y 608.436,Z 364.7,A -85,B 0,C 180,E1 -386.036,E2 -386.036} C_VEL
LIN {X 0,Y 608.464,Z 364.696,A -85,B 0,C 180,E1 -388.624,E2 -388.624} C_VEL
LIN {X 0,Y 608.462,Z 364.697,A -85,B 0,C 180,E1 -391.317,E2 -391.317} C_VEL
LIN {X 0,Y 608.456,Z 364.694,A -85,B 0,C 180,E1 -393.737,E2 -393.737} C_VEL
LIN {X 0,Y 608.459,Z 364.692,A -85,B 0,C 180,E1 -396.092,E2 -396.092} C_VEL
LIN {X 0,Y 608.466,Z 364.692,A -85,B 0,C 180,E1 -398.588,E2 -398.588} C_VEL
LIN {X 0,Y 608.439,Z 364.695,A -85,B 0,C 180,E1 -401.344,E2 -401.344} C_VEL
LIN {X 0,Y 608.457,Z 364.693,A -85,B 0,C 180,E1 -403.871,E2 -403.871} C_VEL
LIN {X 0,Y 608.47,Z 364.691,A -85,B 0,C 180,E1 -406.692,E2 -406.692} C_VEL
LIN {X 0,Y 608.452,Z 364.697,A -85,B 0,C 180,E1 -408.826,E2 -408.826} C_VEL
LIN {X 0,Y 608.461,Z 364.697,A -85,B 0,C 180,E1 -411.414,E2 -411.414} C_VEL
LIN {X 0,Y 608.471,Z 364.695,A -85,B 0,C 180,E1 -413.952,E2 -413.952} C_VEL
LIN {X 0,Y 608.465,Z 364.693,A -85,B 0,C 180,E1 -416.332,E2 -416.332} C_VEL
LIN {X 0,Y 608.469,Z 364.692,A -85,B 0,C 180,E1 -418.729,E2 -418.729} C_VEL
LIN {X 0,Y 608.478,Z 364.744,A -85,B 0,C 180,E1 -420.16,E2 -420.16} C_VEL
LIN {X 0,Y 608.503,Z 376.481,A -85,B 0,C 180,E1 -422.789,E2 -422.789} C_VEL
LIN {X 0,Y 608.463,Z 386.894,A -85,B 0,C 180,E1 -425.067,E2 -425.067} C_VEL
LIN {X 0,Y 608.472,Z 398.67,A -85,B 0,C 180,E1 -427.597,E2 -427.597} C_VEL
LIN {X 0,Y 608.472,Z 412.128,A -85,B 0,C 180,E1 -430.432,E2 -430.432} C_VEL
LIN {X 0,Y 608.479,Z 425.586,A -85,B 0,C 180,E1 -433.219,E2 -433.219} C_VEL
LIN {X 0,Y 608.475,Z 439.13,A -85,B 0,C 180,E1 -435.982,E2 -435.982} C_VEL
LIN {X 0,Y 608.446,Z 450.137,A -85,B 0,C 180,E1 -438.203,E2 -438.203} C_VEL
LIN {X 0,Y 608.538,Z 464.258,A -85,B 0,C 180,E1 -438.468,E2 -438.468} C_VEL
LIN {X 0,Y 608.493,Z 476.101,A -85,B 0,C 180,E1 -438.814,E2 -438.814} C_VEL
LIN {X 0,Y 608.476,Z 487.388,A -85,B 0,C 180,E1 -439.265,E2 -439.265} C_VEL
LIN {X 0,Y 608.496,Z 498.785,A -85,B 0,C 180,E1 -439.857,E2 -439.857} C_VEL
LIN {X 0,Y 608.503,Z 510.276,A -85,B 0,C 180,E1 -440.613,E2 -440.613} C_VEL
LIN {X 0,Y 608.471,Z 519.555,A -85,B 0,C 180,E1 -441.366,E2 -441.366} C_VEL
LIN {X 0,Y 608.455,Z 528.004,A -85,B 0,C 180,E1 -442.201,E2 -442.201} C_VEL
LIN {X 0,Y 608.461,Z 536.247,A -85,B 0,C 180,E1 -443.202,E2 -443.202} C_VEL
LIN {X 0,Y 608.437,Z 542.886,A -85,B 0,C 180,E1 -444.201,E2 -444.201} C_VEL
LIN {X 0,Y 608.432,Z 548.957,A -85,B 0,C 180,E1 -445.364,E2 -445.364} C_VEL
LIN {X 0,Y 608.449,Z 552.901,A -85,B 0,C 180,E1 -446.359,E2 -446.359} C_VEL
LIN {X 0,Y 608.425,Z 555.813,A -85,B 0,C 180,E1 -447.353,E2 -447.353} C_VEL
LIN {X 0,Y 608.444,Z 557.204,A -85,B 0,C 180,E1 -448.016,E2 -448.016} C_VEL
LIN {X 0,Y 608.438,Z 558.784,A -85,B 0,C 180,E1 -449.34,E2 -449.34} C_VEL
LIN {X 0,Y 608.434,Z 559,A -85,B 0,C 180,E1 -450.001,E2 -450.001} C_VEL
LIN {X 0,Y 608.448,Z 558.182,A -85,B 0,C 180,E1 -451.325,E2 -451.325} C_VEL
LIN {X 0,Y 608.444,Z 557.199,A -85,B 0,C 180,E1 -451.987,E2 -451.987} C_VEL
LIN {X 0,Y 608.425,Z 555.805,A -85,B 0,C 180,E1 -452.65,E2 -452.65} C_VEL
LIN {X 0,Y 608.449,Z 552.891,A -85,B 0,C 180,E1 -453.644,E2 -453.644} C_VEL
LIN {X 0,Y 608.432,Z 548.944,A -85,B 0,C 180,E1 -454.639,E2 -454.639} C_VEL
LIN {X 0,Y 608.437,Z 542.868,A -85,B 0,C 180,E1 -455.802,E2 -455.802} C_VEL
LIN {X 0,Y 608.463,Z 536.225,A -85,B 0,C 180,E1 -456.801,E2 -456.801} C_VEL
LIN {X 0,Y 608.456,Z 527.977,A -85,B 0,C 180,E1 -457.801,E2 -457.801} C_VEL
LIN {X 0,Y 608.472,Z 519.521,A -85,B 0,C 180,E1 -458.637,E2 -458.637} C_VEL
LIN {X 0,Y 608.481,Z 509.073,A -85,B 0,C 180,E1 -459.475,E2 -459.475} C_VEL
LIN {X 0,Y 608.5,Z 498.734,A -85,B 0,C 180,E1 -460.146,E2 -460.146} C_VEL
LIN {X 0,Y 608.478,Z 487.336,A -85,B 0,C 180,E1 -460.737,E2 -460.737} C_VEL
LIN {X 0,Y 608.499,Z 474.98,A -85,B 0,C 180,E1 -461.222,E2 -461.222} C_VEL
LIN {X 0,Y 608.548,Z 461.387,A -85,B 0,C 180,E1 -461.598,E2 -461.598} C_VEL
LIN {X 0,Y 608.45,Z 450.07,A -85,B 0,C 180,E1 -461.811,E2 -461.811} C_VEL
LIN {X 0,Y 608.457,Z 437.347,A -85,B 0,C 180,E1 -464.38,E2 -464.38} C_VEL
LIN {X 0,Y 608.468,Z 423.889,A -85,B 0,C 180,E1 -467.131,E2 -467.131} C_VEL
LIN {X 0,Y 608.491,Z 410.431,A -85,B 0,C 180,E1 -469.922,E2 -469.922} C_VEL
LIN {X 0,Y 608.471,Z 396.974,A -85,B 0,C 180,E1 -472.764,E2 -472.764} C_VEL
LIN {X 0,Y 608.5,Z 385.196,A -85,B 0,C 180,E1 -475.3,E2 -475.3} C_VEL
LIN {X 0,Y 608.525,Z 371.738,A -85,B 0,C 180,E1 -478.264,E2 -478.264} C_VEL
LIN {X 0,Y 608.448,Z 364.693,A -85,B 0,C 180,E1 -479.872,E2 -479.872} C_VEL
LIN {X 0,Y 608.451,Z 364.694,A -85,B 0,C 180,E1 -482.52,E2 -482.52} C_VEL
LIN {X 0,Y 608.452,Z 364.694,A -85,B 0,C 180,E1 -484.905,E2 -484.905} C_VEL
LIN {X 0,Y 608.471,Z 364.689,A -85,B 0,C 180,E1 -487.747,E2 -487.747} C_VEL
LIN {X 0,Y 608.438,Z 364.695,A -85,B 0,C 180,E1 -490.327,E2 -490.327} C_VEL
LIN {X 0,Y 608.454,Z 364.694,A -85,B 0,C 180,E1 -493.307,E2 -493.307} C_VEL
LIN {X 0,Y 608.432,Z 364.692,A -85,B 0,C 180,E1 -496.127,E2 -496.127} C_VEL
LIN {X 0,Y 608.448,Z 364.697,A -85,B 0,C 180,E1 -498.823,E2 -498.823} C_VEL
LIN {X 0,Y 608.458,Z 364.689,A -85,B 0,C 180,E1 -501.761,E2 -501.761} C_VEL
LIN {X 0,Y 608.45,Z 364.693,A -85,B 0,C 180,E1 -503.955,E2 -503.955} C_VEL
LIN {X 0,Y 608.447,Z 364.696,A -85,B 0,C 180,E1 -506.328,E2 -506.328} C_VEL
LIN {X 0,Y 608.44,Z 364.691,A -85,B 0,C 180,E1 -508.734,E2 -508.734} C_VEL
LIN {X 0,Y 608.475,Z 364.693,A -85,B 0,C 180,E1 -511.38,E2 -511.38} C_VEL
LIN {X 0,Y 608.404,Z 364.695,A -85,B 0,C 180,E1 -514.293,E2 -514.293} C_VEL
LIN {X 0,Y 608.445,Z 364.699,A -85,B 0,C 180,E1 -516.876,E2 -516.876} C_VEL
LIN {X 0,Y 608.462,Z 364.689,A -85,B 0,C 180,E1 -519.323,E2 -519.323} C_VEL
LIN {X 0,Y 608.446,Z 364.693,A -85,B 0,C 180,E1 -521.828,E2 -521.828} C_VEL
LIN {X 0,Y 608.461,Z 364.69,A -85,B 0,C 180,E1 -524.594,E2 -524.594} C_VEL
LIN {X 0,Y 608.476,Z 364.69,A -85,B 0,C 180,E1 -527.323,E2 -527.323} C_VEL
LIN {X 0,Y 608.418,Z 364.695,A -85,B 0,C 180,E1 -530.022,E2 -530.022} C_VEL
LIN {X 0,Y 608.432,Z 364.696,A -85,B 0,C 180,E1 -532.7,E2 -532.7} C_VEL
LIN {X 0,Y 608.427,Z 364.694,A -85,B 0,C 180,E1 -535.362,E2 -535.362} C_VEL
LIN {X 0,Y 608.426,Z 364.742,A -85,B 0,C 180,E1 -536.357,E2 -536.357} C_VEL
LIN {X 0,Y 608.442,Z 371.12,A -85,B 0,C 180,E1 -538.676,E2 -538.676} C_VEL
LIN {X 0,Y 608.477,Z 376.291,A -85,B 0,C 180,E1 -540.662,E2 -540.662} C_VEL
LIN {X 0,Y 608.444,Z 382.608,A -85,B 0,C 180,E1 -543.311,E2 -543.311} C_VEL
LIN {X 0,Y 608.468,Z 389.091,A -85,B 0,C 180,E1 -545.967,E2 -545.967} C_VEL
LIN {X 0,Y 608.447,Z 395.755,A -85,B 0,C 180,E1 -548.636,E2 -548.636} C_VEL
LIN {X 0,Y 608.431,Z 397.568,A -85,B 0,C 180,E1 -549.353,E2 -549.353} C_VEL
LIN {X 0,Y 607.77,Z 398.99,A -85,B 0,C 180,E1 -549.889,E2 -549.889} C_VEL
LIN {X 0,Y 604.919,Z 401.451,A -85,B 0,C 180,E1 -550.756,E2 -550.756} C_VEL
LIN {X 0,Y 602.496,Z 403.434,A -85,B 0,C 180,E1 -551.452,E2 -551.452} C_VEL
LIN {X 0,Y 601.44,Z 404.896,A -85,B 0,C 180,E1 -551.991,E2 -551.991} C_VEL
LIN {X 0,Y 601.346,Z 405.37,A -85,B 0,C 180,E1 -552.174,E2 -552.174} C_VEL
LIN {X 0,Y 601.356,Z 412.371,A -85,B 0,C 180,E1 -554.899,E2 -554.899} C_VEL
LIN {X 0,Y 601.328,Z 419.647,A -85,B 0,C 180,E1 -557.69,E2 -557.69} C_VEL
LIN {X 0,Y 601.349,Z 423.471,A -85,B 0,C 180,E1 -559.145,E2 -559.145} C_VEL
LIN {X 0,Y 601.601,Z 430.548,A -85,B 0,C 180,E1 -559.292,E2 -559.292} C_VEL
LIN {X 0,Y 601.537,Z 443.013,A -85,B 0,C 180,E1 -559.627,E2 -559.627} C_VEL
LIN {X 0,Y 601.521,Z 454.802,A -85,B 0,C 180,E1 -560.072,E2 -560.072} C_VEL
LIN {X 0,Y 601.501,Z 467.011,A -85,B 0,C 180,E1 -560.678,E2 -560.678} C_VEL
LIN {X 0,Y 601.474,Z 478.491,A -85,B 0,C 180,E1 -561.416,E2 -561.416} C_VEL
LIN {X 0,Y 601.438,Z 488.612,A -85,B 0,C 180,E1 -562.226,E2 -562.226} C_VEL
LIN {X 0,Y 601.413,Z 497.006,A -85,B 0,C 180,E1 -563.046,E2 -563.046} C_VEL
LIN {X 0,Y 601.398,Z 504.715,A -85,B 0,C 180,E1 -563.959,E2 -563.959} C_VEL
LIN {X 0,Y 601.387,Z 512.204,A -85,B 0,C 180,E1 -565.064,E2 -565.064} C_VEL
LIN {X 0,Y 601.365,Z 517.671,A -85,B 0,C 180,E1 -566.08,E2 -566.08} C_VEL
LIN {X 0,Y 601.336,Z 522.02,A -85,B 0,C 180,E1 -567.116,E2 -567.116} C_VEL
LIN {X 0,Y 601.355,Z 524.498,A -85,B 0,C 180,E1 -567.87,E2 -567.87} C_VEL
LIN {X 0,Y 601.339,Z 526.688,A -85,B 0,C 180,E1 -568.771,E2 -568.771} C_VEL
LIN {X 0,Y 601.341,Z 527.794,A -85,B 0,C 180,E1 -569.397,E2 -569.397} C_VEL
LIN {X 0,Y 601.344,Z 528.64,A -85,B 0,C 180,E1 -570.168,E2 -570.168} C_VEL
LIN {X 0,Y 601.33,Z 528.915,A -85,B 0,C 180,E1 -571.44,E2 -571.44} C_VEL
LIN {X 0,Y 601.335,Z 527.78,A -85,B 0,C 180,E1 -572.702,E2 -572.702} C_VEL
LIN {X 0,Y 601.338,Z 525.291,A -85,B 0,C 180,E1 -573.922,E2 -573.922} C_VEL
LIN {X 0,Y 601.331,Z 521.543,A -85,B 0,C 180,E1 -575.103,E2 -575.103} C_VEL
LIN {X 0,Y 601.365,Z 516.493,A -85,B 0,C 180,E1 -576.255,E2 -576.255} C_VEL
LIN {X 0,Y 601.374,Z 510.043,A -85,B 0,C 180,E1 -577.374,E2 -577.374} C_VEL
LIN {X 0,Y 601.384,Z 502.063,A -85,B 0,C 180,E1 -578.464,E2 -578.464} C_VEL
LIN {X 0,Y 601.438,Z 494.295,A -85,B 0,C 180,E1 -579.326,E2 -579.326} C_VEL
LIN {X 0,Y 601.435,Z 484.618,A -85,B 0,C 180,E1 -580.204,E2 -580.204} C_VEL
LIN {X 0,Y 601.428,Z 473.995,A -85,B 0,C 180,E1 -580.984,E2 -580.984} C_VEL
LIN {X 0,Y 601.439,Z 463.681,A -85,B 0,C 180,E1 -581.594,E2 -581.594} C_VEL
LIN {X 0,Y 601.477,Z 451.644,A -85,B 0,C 180,E1 -582.154,E2 -582.154} C_VEL
LIN {X 0,Y 601.552,Z 438.884,A -85,B 0,C 180,E1 -582.589,E2 -582.589} C_VEL
LIN {X 0,Y 601.595,Z 425.896,A -85,B 0,C 180,E1 -582.888,E2 -582.888} C_VEL
LIN {X 0,Y 601.329,Z 423.429,A -85,B 0,C 180,E1 -582.961,E2 -582.961} C_VEL
LIN {X 0,Y 601.295,Z 416.831,A -85,B 0,C 180,E1 -585.477,E2 -585.477} C_VEL
LIN {X 0,Y 601.318,Z 409.705,A -85,B 0,C 180,E1 -588.225,E2 -588.225} C_VEL
LIN {X 0,Y 601.332,Z 402.955,A -85,B 0,C 180,E1 -590.867,E2 -590.867} C_VEL
LIN {X 0,Y 601.339,Z 395.721,A -85,B 0,C 180,E1 -593.747,E2 -593.747} C_VEL
LIN {X 0,Y 601.37,Z 389.987,A -85,B 0,C 180,E1 -596.073,E2 -596.073} C_VEL
LIN {X 0,Y 601.39,Z 384,A -85,B 0,C 180,E1 -598.55,E2 -598.55} C_VEL
LIN {X 0,Y 601.395,Z 377.237,A -85,B 0,C 180,E1 -601.37,E2 -601.37} C_VEL
LIN {X 0,Y 601.42,Z 369.633,A -85,B 0,C 180,E1 -604.381,E2 -604.381} C_VEL
LIN {X 0,Y 601.439,Z 365.568,A -85,B 0,C 180,E1 -606.041,E2 -606.041} C_VEL
LIN {X 0,Y 601.403,Z 365.574,A -85,B 0,C 180,E1 -608.76,E2 -608.76} C_VEL
LIN {X 0,Y 601.383,Z 365.574,A -85,B 0,C 180,E1 -611.606,E2 -611.606} C_VEL
LIN {X 0,Y 601.413,Z 365.568,A -85,B 0,C 180,E1 -614.408,E2 -614.408} C_VEL
LIN {X 0,Y 601.406,Z 365.571,A -85,B 0,C 180,E1 -617.17,E2 -617.17} C_VEL
LIN {X 0,Y 601.43,Z 365.573,A -85,B 0,C 180,E1 -619.904,E2 -619.904} C_VEL
LIN {X 0,Y 601.443,Z 365.567,A -85,B 0,C 180,E1 -622.614,E2 -622.614} C_VEL
LIN {X 0,Y 601.393,Z 365.571,A -85,B 0,C 180,E1 -625.306,E2 -625.306} C_VEL
LIN {X 0,Y 601.435,Z 365.568,A -85,B 0,C 180,E1 -627.99,E2 -627.99} C_VEL
LIN {X 0,Y 601.439,Z 365.612,A -85,B 0,C 180,E1 -630.584,E2 -630.584} C_VEL
LIN {X 0,Y 601.4,Z 371.636,A -85,B 0,C 180,E1 -633.348,E2 -633.348} C_VEL
LIN {X 0,Y 601.401,Z 377.536,A -85,B 0,C 180,E1 -636.036,E2 -636.036} C_VEL
LIN {X 0,Y 601.375,Z 383.64,A -85,B 0,C 180,E1 -638.737,E2 -638.737} C_VEL
LIN {X 0,Y 601.375,Z 389.918,A -85,B 0,C 180,E1 -641.457,E2 -641.457} C_VEL
LIN {X 0,Y 601.364,Z 396.379,A -85,B 0,C 180,E1 -644.205,E2 -644.205} C_VEL
LIN {X 0,Y 601.347,Z 403.028,A -85,B 0,C 180,E1 -646.986,E2 -646.986} C_VEL
LIN {X 0,Y 601.321,Z 409.875,A -85,B 0,C 180,E1 -649.81,E2 -649.81} C_VEL
LIN {X 0,Y 601.303,Z 416.927,A -85,B 0,C 180,E1 -652.685,E2 -652.685} C_VEL
LIN {X 0,Y 601.351,Z 419.336,A -85,B 0,C 180,E1 -653.662,E2 -653.662} C_VEL
LIN {X 0,Y 601.476,Z 431.367,A -85,B 0,C 180,E1 -654,E2 -654} C_VEL
LIN {X 0,Y 601.415,Z 441.213,A -85,B 0,C 180,E1 -654.383,E2 -654.383} C_VEL
LIN {X 0,Y 601.377,Z 449.397,A -85,B 0,C 180,E1 -654.795,E2 -654.795} C_VEL
LIN {X 0,Y 601.389,Z 458.026,A -85,B 0,C 180,E1 -655.339,E2 -655.339} C_VEL
LIN {X 0,Y 601.418,Z 465.61,A -85,B 0,C 180,E1 -655.928,E2 -655.928} C_VEL
LIN {X 0,Y 601.367,Z 474.049,A -85,B 0,C 180,E1 -656.737,E2 -656.737} C_VEL
LIN {X 0,Y 601.391,Z 480.915,A -85,B 0,C 180,E1 -657.58,E2 -657.58} C_VEL
LIN {X 0,Y 601.356,Z 486.48,A -85,B 0,C 180,E1 -658.438,E2 -658.438} C_VEL
LIN {X 0,Y 601.349,Z 491.311,A -85,B 0,C 180,E1 -659.394,E2 -659.394} C_VEL
LIN {X 0,Y 601.339,Z 494.257,A -85,B 0,C 180,E1 -660.166,E2 -660.166} C_VEL
LIN {X 0,Y 601.332,Z 496.465,A -85,B 0,C 180,E1 -660.944,E2 -660.944} C_VEL
LIN {X 0,Y 601.333,Z 497.968,A -85,B 0,C 180,E1 -661.728,E2 -661.728} C_VEL
LIN {X 0,Y 601.338,Z 498.866,A -85,B 0,C 180,E1 -662.703,E2 -662.703} C_VEL
LIN {X 0,Y 601.319,Z 498.575,A -85,B 0,C 180,E1 -663.92,E2 -663.92} C_VEL
LIN {X 0,Y 601.322,Z 496.568,A -85,B 0,C 180,E1 -665.102,E2 -665.102} C_VEL
LIN {X 0,Y 601.329,Z 494.831,A -85,B 0,C 180,E1 -665.756,E2 -665.756} C_VEL
LIN {X 0,Y 601.352,Z 491.817,A -85,B 0,C 180,E1 -666.584,E2 -666.584} C_VEL
LIN {X 0,Y 601.346,Z 486.587,A -85,B 0,C 180,E1 -667.634,E2 -667.634} C_VEL
LIN {X 0,Y 601.363,Z 481.244,A -85,B 0,C 180,E1 -668.463,E2 -668.463} C_VEL
LIN {X 0,Y 601.377,Z 474.26,A -85,B 0,C 180,E1 -669.33,E2 -669.33} C_VEL
LIN {X 0,Y 601.408,Z 466.383,A -85,B 0,C 180,E1 -670.098,E2 -670.098} C_VEL
LIN {X 0,Y 601.399,Z 457.678,A -85,B 0,C 180,E1 -670.775,E2 -670.775} C_VEL
LIN {X 0,Y 601.417,Z 449.029,A -85,B 0,C 180,E1 -671.315,E2 -671.315} C_VEL
LIN {X 0,Y 601.475,Z 438.855,A -85,B 0,C 180,E1 -671.814,E2 -671.814} C_VEL
LIN {X 0,Y 601.484,Z 427.1,A -85,B 0,C 180,E1 -672.222,E2 -672.222} C_VEL
LIN {X 0,Y 601.312,Z 419.325,A -85,B 0,C 180,E1 -672.433,E2 -672.433} C_VEL
LIN {X 0,Y 601.313,Z 413.013,A -85,B 0,C 180,E1 -674.997,E2 -674.997} C_VEL
LIN {X 0,Y 601.361,Z 407.12,A -85,B 0,C 180,E1 -677.411,E2 -677.411} C_VEL
LIN {X 0,Y 601.313,Z 399.74,A -85,B 0,C 180,E1 -680.475,E2 -680.475} C_VEL
LIN {X 0,Y 601.29,Z 394.618,A -85,B 0,C 180,E1 -682.632,E2 -682.632} C_VEL
LIN {X 0,Y 601.356,Z 388.915,A -85,B 0,C 180,E1 -685.064,E2 -685.064} C_VEL
LIN {X 0,Y 601.36,Z 381.553,A -85,B 0,C 180,E1 -688.271,E2 -688.271} C_VEL
LIN {X 0,Y 601.422,Z 374.613,A -85,B 0,C 180,E1 -691.373,E2 -691.373} C_VEL
LIN {X 0,Y 601.41,Z 368.571,A -85,B 0,C 180,E1 -694.127,E2 -694.127} C_VEL
LIN {X 0,Y 601.426,Z 365.571,A -85,B 0,C 180,E1 -695.534,E2 -695.534} C_VEL
LIN {X 0,Y 601.411,Z 365.574,A -85,B 0,C 180,E1 -698.041,E2 -698.041} C_VEL
LIN {X 0,Y 601.415,Z 365.572,A -85,B 0,C 180,E1 -700.901,E2 -700.901} C_VEL
LIN {X 0,Y 601.419,Z 365.57,A -85,B 0,C 180,E1 -703.713,E2 -703.713} C_VEL
LIN {X 0,Y 601.404,Z 365.572,A -85,B 0,C 180,E1 -706.484,E2 -706.484} C_VEL
LIN {X 0,Y 601.425,Z 365.569,A -85,B 0,C 180,E1 -709.224,E2 -709.224} C_VEL
LIN {X 0,Y 601.419,Z 365.569,A -85,B 0,C 180,E1 -711.939,E2 -711.939} C_VEL
LIN {X 0,Y 601.422,Z 365.569,A -85,B 0,C 180,E1 -714.636,E2 -714.636} C_VEL
LIN {X 0,Y 601.435,Z 365.568,A -85,B 0,C 180,E1 -717.321,E2 -717.321} C_VEL
LIN {X 0,Y 601.418,Z 365.57,A -85,B 0,C 180,E1 -720,E2 -720} C_VEL
LIN {X 0,Y 601.433,Z 365.568,A -85,B 0,C 180,E1 -722.679,E2 -722.679} C_VEL
LIN {X 0,Y 601.424,Z 365.569,A -85,B 0,C 180,E1 -725.364,E2 -725.364} C_VEL
LIN {X 0,Y 601.42,Z 365.569,A -85,B 0,C 180,E1 -728.061,E2 -728.061} C_VEL
LIN {X 0,Y 601.462,Z 365.566,A -85,B 0,C 180,E1 -731.045,E2 -731.045} C_VEL
LIN {X 0,Y 601.438,Z 365.569,A -85,B 0,C 180,E1 -734.205,E2 -734.205} C_VEL
LIN {X 0,Y 601.418,Z 365.571,A -85,B 0,C 180,E1 -736.987,E2 -736.987} C_VEL
LIN {X 0,Y 601.392,Z 365.573,A -85,B 0,C 180,E1 -739.81,E2 -739.81} C_VEL
LIN {X 0,Y 601.436,Z 365.567,A -85,B 0,C 180,E1 -742.682,E2 -742.682} C_VEL
LIN {X 0,Y 601.382,Z 365.577,A -85,B 0,C 180,E1 -744.88,E2 -744.88} C_VEL
LIN {X 0,Y 601.408,Z 365.576,A -85,B 0,C 180,E1 -747.367,E2 -747.367} C_VEL
LIN {X 0,Y 601.429,Z 365.571,A -85,B 0,C 180,E1 -750.164,E2 -750.164} C_VEL
LIN {X 0,Y 601.41,Z 365.575,A -85,B 0,C 180,E1 -752.719,E2 -752.719} C_VEL
LIN {X 0,Y 601.407,Z 365.573,A -85,B 0,C 180,E1 -755.118,E2 -755.118} C_VEL
LIN {X 0,Y 601.417,Z 365.57,A -85,B 0,C 180,E1 -757.421,E2 -757.421} C_VEL
LIN {X 0,Y 601.4,Z 365.572,A -85,B 0,C 180,E1 -759.996,E2 -759.996} C_VEL
LIN {X 0,Y 601.428,Z 365.568,A -85,B 0,C 180,E1 -762.669,E2 -762.669} C_VEL
LIN {X 0,Y 601.411,Z 365.571,A -85,B 0,C 180,E1 -765.484,E2 -765.484} C_VEL
LIN {X 0,Y 601.419,Z 365.571,A -85,B 0,C 180,E1 -768.408,E2 -768.408} C_VEL
LIN {X 0,Y 601.428,Z 365.569,A -85,B 0,C 180,E1 -770.878,E2 -770.878} C_VEL
LIN {X 0,Y 601.433,Z 365.569,A -85,B 0,C 180,E1 -773.736,E2 -773.736} C_VEL
LIN {X 0,Y 601.431,Z 365.568,A -85,B 0,C 180,E1 -776.065,E2 -776.065} C_VEL
LIN {X 0,Y 601.423,Z 365.571,A -85,B 0,C 180,E1 -779.061,E2 -779.061} C_VEL
LIN {X 0,Y 601.455,Z 365.635,A -85,B 0,C 180,E1 -779.98,E2 -779.98} C_VEL
LIN {X 0,Y 601.559,Z 371.753,A -85,B 0,C 180,E1 -781.382,E2 -781.382} C_VEL
LIN {X 0,Y 601.561,Z 383.915,A -85,B 0,C 180,E1 -784.104,E2 -784.104} C_VEL
LIN {X 0,Y 601.471,Z 396.987,A -85,B 0,C 180,E1 -786.958,E2 -786.958} C_VEL
LIN {X 0,Y 601.469,Z 408.763,A -85,B 0,C 180,E1 -789.482,E2 -789.482} C_VEL
LIN {X 0,Y 601.425,Z 422.222,A -85,B 0,C 180,E1 -792.315,E2 -792.315} C_VEL
LIN {X 0,Y 601.435,Z 433.998,A -85,B 0,C 180,E1 -794.758,E2 -794.758} C_VEL
LIN {X 0,Y 601.374,Z 445.774,A -85,B 0,C 180,E1 -797.173,E2 -797.173} C_VEL
LIN {X 0,Y 601.409,Z 450.085,A -85,B 0,C 180,E1 -798.052,E2 -798.052} C_VEL
LIN {X 0,Y 601.604,Z 464.257,A -85,B 0,C 180,E1 -798.333,E2 -798.333} C_VEL
LIN {X 0,Y 601.541,Z 476.797,A -85,B 0,C 180,E1 -798.708,E2 -798.708} C_VEL
LIN {X 0,Y 601.482,Z 489.211,A -85,B 0,C 180,E1 -799.227,E2 -799.227} C_VEL
LIN {X 0,Y 601.474,Z 501.609,A -85,B 0,C 180,E1 -799.907,E2 -799.907} C_VEL
LIN {X 0,Y 601.449,Z 512.497,A -85,B 0,C 180,E1 -800.671,E2 -800.671} C_VEL
LIN {X 0,Y 601.428,Z 523.13,A -85,B 0,C 180,E1 -801.603,E2 -801.603} C_VEL
LIN {X 0,Y 601.417,Z 530.975,A -85,B 0,C 180,E1 -802.447,E2 -802.447} C_VEL
LIN {X 0,Y 601.369,Z 538.233,A -85,B 0,C 180,E1 -803.399,E2 -803.399} C_VEL
LIN {X 0,Y 601.371,Z 543.875,A -85,B 0,C 180,E1 -804.301,E2 -804.301} C_VEL
LIN {X 0,Y 601.336,Z 548.957,A -85,B 0,C 180,E1 -805.309,E2 -805.309} C_VEL
LIN {X 0,Y 601.368,Z 552.901,A -85,B 0,C 180,E1 -806.316,E2 -806.316} C_VEL
LIN {X 0,Y 601.325,Z 555.813,A -85,B 0,C 180,E1 -807.322,E2 -807.322} C_VEL
LIN {X 0,Y 601.343,Z 557.204,A -85,B 0,C 180,E1 -807.992,E2 -807.992} C_VEL
LIN {X 0,Y 601.339,Z 558.785,A -85,B 0,C 180,E1 -809.332,E2 -809.332} C_VEL
LIN {X 0,Y 601.335,Z 559,A -85,B 0,C 180,E1 -810.001,E2 -810.001} C_VEL
LIN {X 0,Y 601.347,Z 558.182,A -85,B 0,C 180,E1 -811.341,E2 -811.341} C_VEL
LIN {X 0,Y 601.343,Z 557.199,A -85,B 0,C 180,E1 -812.011,E2 -812.011} C_VEL
LIN {X 0,Y 601.325,Z 555.805,A -85,B 0,C 180,E1 -812.681,E2 -812.681} C_VEL
LIN {X 0,Y 601.368,Z 552.891,A -85,B 0,C 180,E1 -813.687,E2 -813.687} C_VEL
LIN {X 0,Y 601.336,Z 548.944,A -85,B 0,C 180,E1 -814.694,E2 -814.694} C_VEL
LIN {X 0,Y 601.372,Z 542.869,A -85,B 0,C 180,E1 -815.871,E2 -815.871} C_VEL
LIN {X 0,Y 601.383,Z 536.226,A -85,B 0,C 180,E1 -816.881,E2 -816.881} C_VEL
LIN {X 0,Y 601.401,Z 527.978,A -85,B 0,C 180,E1 -817.894,E2 -817.894} C_VEL
LIN {X 0,Y 601.437,Z 519.522,A -85,B 0,C 180,E1 -818.739,E2 -818.739} C_VEL
LIN {X 0,Y 601.451,Z 509.075,A -85,B 0,C 180,E1 -819.586,E2 -819.586} C_VEL
LIN {X 0,Y 601.49,Z 498.736,A -85,B 0,C 180,E1 -820.265,E2 -820.265} C_VEL
LIN {X 0,Y 601.493,Z 487.116,A -85,B 0,C 180,E1 -820.874,E2 -820.874} C_VEL
LIN {X 0,Y 601.528,Z 474.283,A -85,B 0,C 180,E1 -821.377,E2 -821.377} C_VEL
LIN {X 0,Y 601.594,Z 461.387,A -85,B 0,C 180,E1 -821.734,E2 -821.734} C_VEL
LIN {X 0,Y 601.41,Z 450.07,A -85,B 0,C 180,E1 -821.951,E2 -821.951} C_VEL
LIN {X 0,Y 601.396,Z 437.347,A -85,B 0,C 180,E1 -824.553,E2 -824.553} C_VEL
LIN {X 0,Y 601.429,Z 423.889,A -85,B 0,C 180,E1 -827.337,E2 -827.337} C_VEL
LIN {X 0,Y 601.474,Z 412.113,A -85,B 0,C 180,E1 -829.808,E2 -829.808} C_VEL
LIN {X 0,Y 601.491,Z 398.655,A -85,B 0,C 180,E1 -832.681,E2 -832.681} C_VEL
LIN {X 0,Y 601.509,Z 386.879,A -85,B 0,C 180,E1 -835.244,E2 -835.244} C_VEL
LIN {X 0,Y 601.604,Z 375.103,A -85,B 0,C 180,E1 -837.859,E2 -837.859} C_VEL
LIN {X 0,Y 601.587,Z 366.738,A -85,B 0,C 180,E1 -839.759,E2 -839.759} C_VEL
LIN {X 0,Y 601.404,Z 365.571,A -85,B 0,C 180,E1 -840.08,E2 -840.08} C_VEL
LIN {X 0,Y 601.416,Z 365.573,A -85,B 0,C 180,E1 -842.714,E2 -842.714} C_VEL
LIN {X 0,Y 601.402,Z 365.57,A -85,B 0,C 180,E1 -845.112,E2 -845.112} C_VEL
LIN {X 0,Y 601.437,Z 365.564,A -85,B 0,C 180,E1 -847.42,E2 -847.42} C_VEL
LIN {X 0,Y 601.405,Z 365.576,A -85,B 0,C 180,E1 -849.996,E2 -849.996} C_VEL
LIN {X 0,Y 601.358,Z 365.573,A -85,B 0,C 180,E1 -852.676,E2 -852.676} C_VEL
LIN {X 0,Y 601.404,Z 365.574,A -85,B 0,C 180,E1 -855.48,E2 -855.48} C_VEL
LIN {X 0,Y 601.413,Z 365.568,A -85,B 0,C 180,E1 -858.409,E2 -858.409} C_VEL
LIN {X 0,Y 601.407,Z 365.574,A -85,B 0,C 180,E1 -860.873,E2 -860.873} C_VEL
LIN {X 0,Y 601.404,Z 365.567,A -85,B 0,C 180,E1 -863.417,E2 -863.417} C_VEL
LIN {X 0,Y 601.421,Z 365.573,A -85,B 0,C 180,E1 -866.067,E2 -866.067} C_VEL
LIN {X 0,Y 601.416,Z 365.567,A -85,B 0,C 180,E1 -868.547,E2 -868.547} C_VEL
LIN {X 0,Y 601.431,Z 365.571,A -85,B 0,C 180,E1 -871.373,E2 -871.373} C_VEL
LIN {X 0,Y 601.361,Z 365.573,A -85,B 0,C 180,E1 -874.379,E2 -874.379} C_VEL
LIN {X 0,Y 601.382,Z 365.574,A -85,B 0,C 180,E1 -876.588,E2 -876.588} C_VEL
LIN {X 0,Y 601.423,Z 365.565,A -85,B 0,C 180,E1 -879.478,E2 -879.478} C_VEL
LIN {X 0,Y 601.394,Z 365.577,A -85,B 0,C 180,E1 -882.311,E2 -882.311} C_VEL
LIN {X 0,Y 601.408,Z 365.57,A -85,B 0,C 180,E1 -884.408,E2 -884.408} C_VEL
LIN {X 0,Y 601.418,Z 365.568,A -85,B 0,C 180,E1 -887.172,E2 -887.172} C_VEL
LIN {X 0,Y 601.385,Z 365.572,A -85,B 0,C 180,E1 -889.904,E2 -889.904} C_VEL
LIN {X 0,Y 601.377,Z 365.574,A -85,B 0,C 180,E1 -892.614,E2 -892.614} C_VEL
LIN {X 0,Y 601.399,Z 365.57,A -85,B 0,C 180,E1 -895.308,E2 -895.308} C_VEL
LIN {X 0,Y 601.381,Z 365.709,A -85,B 0,C 180,E1 -896.482,E2 -896.482} C_VEL
LIN {X 0,Y 601.375,Z 371.679,A -85,B 0,C 180,E1 -898.66,E2 -898.66} C_VEL
LIN {X 0,Y 601.419,Z 377.067,A -85,B 0,C 180,E1 -900.669,E2 -900.669} C_VEL
LIN {X 0,Y 601.39,Z 383.544,A -85,B 0,C 180,E1 -903.35,E2 -903.35} C_VEL
LIN {X 0,Y 601.403,Z 390.032,A -85,B 0,C 180,E1 -906.037,E2 -906.037} C_VEL
LIN {X 0,Y 601.374,Z 396.702,A -85,B 0,C 180,E1 -908.738,E2 -908.738} C_VEL
LIN {X 0,Y 601.378,Z 403.549,A -85,B 0,C 180,E1 -911.459,E2 -911.459} C_VEL
LIN {X 0,Y 601.346,Z 405.37,A -85,B 0,C 180,E1 -912.174,E2 -912.174} C_VEL
LIN {X 0,Y 600.653,Z 406.811,A -85,B 0,C 180,E1 -912.716,E2 -912.716} C_VEL
LIN {X 0,Y 597.776,Z 409.277,A -85,B 0,C 180,E1 -913.592,E2 -913.592} C_VEL
LIN {X 0,Y 595.368,Z 411.26,A -85,B 0,C 180,E1 -914.297,E2 -914.297} C_VEL
LIN {X 0,Y 594.347,Z 412.728,A -85,B 0,C 180,E1 -914.842,E2 -914.842} C_VEL
LIN {X 0,Y 594.27,Z 413.206,A -85,B 0,C 180,E1 -915.027,E2 -915.027} C_VEL
LIN {X 0,Y 594.247,Z 418.791,A -85,B 0,C 180,E1 -917.197,E2 -917.197} C_VEL
LIN {X 0,Y 594.262,Z 423.497,A -85,B 0,C 180,E1 -919.011,E2 -919.011} C_VEL
LIN {X 0,Y 594.659,Z 428.561,A -85,B 0,C 180,E1 -919.112,E2 -919.112} C_VEL
LIN {X 0,Y 594.619,Z 442.044,A -85,B 0,C 180,E1 -919.46,E2 -919.46} C_VEL
LIN {X 0,Y 594.507,Z 454.16,A -85,B 0,C 180,E1 -919.914,E2 -919.914} C_VEL
LIN {X 0,Y 594.511,Z 466.022,A -85,B 0,C 180,E1 -920.5,E2 -920.5} C_VEL
LIN {X 0,Y 594.465,Z 476.727,A -85,B 0,C 180,E1 -921.173,E2 -921.173} C_VEL
LIN {X 0,Y 594.399,Z 487.796,A -85,B 0,C 180,E1 -922.049,E2 -922.049} C_VEL
LIN {X 0,Y 594.373,Z 497.141,A -85,B 0,C 180,E1 -922.967,E2 -922.967} C_VEL
LIN {X 0,Y 594.32,Z 504.837,A -85,B 0,C 180,E1 -923.892,E2 -923.892} C_VEL
LIN {X 0,Y 594.297,Z 512.309,A -85,B 0,C 180,E1 -925.009,E2 -925.009} C_VEL
LIN {X 0,Y 594.29,Z 517.591,A -85,B 0,C 180,E1 -926.003,E2 -926.003} C_VEL
LIN {X 0,Y 594.239,Z 522.083,A -85,B 0,C 180,E1 -927.086,E2 -927.086} C_VEL
LIN {X 0,Y 594.233,Z 525.555,A -85,B 0,C 180,E1 -928.234,E2 -928.234} C_VEL
LIN {X 0,Y 594.253,Z 527.192,A -85,B 0,C 180,E1 -929.005,E2 -929.005} C_VEL
LIN {X 0,Y 594.241,Z 528.74,A -85,B 0,C 180,E1 -930.303,E2 -930.303} C_VEL
LIN {X 0,Y 594.228,Z 528.855,A -85,B 0,C 180,E1 -931.619,E2 -931.619} C_VEL
LIN {X 0,Y 594.25,Z 527.396,A -85,B 0,C 180,E1 -932.958,E2 -932.958} C_VEL
LIN {X 0,Y 594.265,Z 524.86,A -85,B 0,C 180,E1 -934.121,E2 -934.121} C_VEL
LIN {X 0,Y 594.253,Z 520.533,A -85,B 0,C 180,E1 -935.415,E2 -935.415} C_VEL
LIN {X 0,Y 594.285,Z 515.706,A -85,B 0,C 180,E1 -936.47,E2 -936.47} C_VEL
LIN {X 0,Y 594.289,Z 509.089,A -85,B 0,C 180,E1 -937.595,E2 -937.595} C_VEL
LIN {X 0,Y 594.33,Z 502.194,A -85,B 0,C 180,E1 -938.537,E2 -938.537} C_VEL
LIN {X 0,Y 594.361,Z 493.951,A -85,B 0,C 180,E1 -939.462,E2 -939.462} C_VEL
LIN {X 0,Y 594.422,Z 484.174,A -85,B 0,C 180,E1 -940.35,E2 -940.35} C_VEL
LIN {X 0,Y 594.428,Z 473.842,A -85,B 0,C 180,E1 -941.113,E2 -941.113} C_VEL
LIN {X 0,Y 594.443,Z 462.358,A -85,B 0,C 180,E1 -941.791,E2 -941.791} C_VEL
LIN {X 0,Y 594.508,Z 449.676,A -85,B 0,C 180,E1 -942.363,E2 -942.363} C_VEL
LIN {X 0,Y 594.633,Z 436.143,A -85,B 0,C 180,E1 -942.803,E2 -942.803} C_VEL
LIN {X 0,Y 594.557,Z 425.62,A -85,B 0,C 180,E1 -943.036,E2 -943.036} C_VEL
LIN {X 0,Y 594.228,Z 423.442,A -85,B 0,C 180,E1 -943.101,E2 -943.101} C_VEL
LIN {X 0,Y 594.236,Z 416.581,A -85,B 0,C 180,E1 -945.749,E2 -945.749} C_VEL
LIN {X 0,Y 594.238,Z 409.484,A -85,B 0,C 180,E1 -948.523,E2 -948.523} C_VEL
LIN {X 0,Y 594.267,Z 402.773,A -85,B 0,C 180,E1 -951.185,E2 -951.185} C_VEL
LIN {X 0,Y 594.296,Z 395.383,A -85,B 0,C 180,E1 -954.17,E2 -954.17} C_VEL
LIN {X 0,Y 594.289,Z 388.424,A -85,B 0,C 180,E1 -957.043,E2 -957.043} C_VEL
LIN {X 0,Y 594.35,Z 382.154,A -85,B 0,C 180,E1 -959.678,E2 -959.678} C_VEL
LIN {X 0,Y 594.335,Z 375.113,A -85,B 0,C 180,E1 -962.536,E2 -962.536} C_VEL
LIN {X 0,Y 594.339,Z 369.394,A -85,B 0,C 180,E1 -964.804,E2 -964.804} C_VEL
LIN {X 0,Y 594.4,Z 366.446,A -85,B 0,C 180,E1 -966.018,E2 -966.018} C_VEL
LIN {X 0,Y 594.39,Z 366.446,A -85,B 0,C 180,E1 -969.223,E2 -969.223} C_VEL
LIN {X 0,Y 594.336,Z 366.456,A -85,B 0,C 180,E1 -972.093,E2 -972.093} C_VEL
LIN {X 0,Y 594.368,Z 366.446,A -85,B 0,C 180,E1 -974.218,E2 -974.218} C_VEL
LIN {X 0,Y 594.387,Z 366.445,A -85,B 0,C 180,E1 -976.32,E2 -976.32} C_VEL
LIN {X 0,Y 594.363,Z 366.447,A -85,B 0,C 180,E1 -979.093,E2 -979.093} C_VEL
LIN {X 0,Y 594.416,Z 366.442,A -85,B 0,C 180,E1 -981.842,E2 -981.842} C_VEL
LIN {X 0,Y 594.389,Z 366.45,A -85,B 0,C 180,E1 -984.571,E2 -984.571} C_VEL
LIN {X 0,Y 594.384,Z 366.446,A -85,B 0,C 180,E1 -987.288,E2 -987.288} C_VEL
LIN {X 0,Y 594.416,Z 366.441,A -85,B 0,C 180,E1 -989.998,E2 -989.998} C_VEL
LIN {X 0,Y 594.411,Z 366.52,A -85,B 0,C 180,E1 -990.591,E2 -990.591} C_VEL
LIN {X 0,Y 594.409,Z 371.107,A -85,B 0,C 180,E1 -992.709,E2 -992.709} C_VEL
LIN {X 0,Y 594.384,Z 376.97,A -85,B 0,C 180,E1 -995.426,E2 -995.426} C_VEL
LIN {X 0,Y 594.339,Z 383.024,A -85,B 0,C 180,E1 -998.156,E2 -998.156} C_VEL
LIN {X 0,Y 594.324,Z 389.582,A -85,B 0,C 180,E1 -1001.042,E2 -1001.042} C_VEL
LIN {X 0,Y 594.294,Z 396.766,A -85,B 0,C 180,E1 -1004.138,E2 -1004.138} C_VEL
LIN {X 0,Y 594.281,Z 403.991,A -85,B 0,C 180,E1 -1007.195,E2 -1007.195} C_VEL
LIN {X 0,Y 594.224,Z 410.858,A -85,B 0,C 180,E1 -1010.057,E2 -1010.057} C_VEL
LIN {X 0,Y 594.216,Z 417.928,A -85,B 0,C 180,E1 -1012.971,E2 -1012.971} C_VEL
LIN {X 0,Y 594.283,Z 419.57,A -85,B 0,C 180,E1 -1013.568,E2 -1013.568} C_VEL
LIN {X 0,Y 594.459,Z 431.146,A -85,B 0,C 180,E1 -1013.884,E2 -1013.884} C_VEL
LIN {X 0,Y 594.403,Z 440.728,A -85,B 0,C 180,E1 -1014.257,E2 -1014.257} C_VEL
LIN {X 0,Y 594.344,Z 449.898,A -85,B 0,C 180,E1 -1014.725,E2 -1014.725} C_VEL
LIN {X 0,Y 594.343,Z 458.588,A -85,B 0,C 180,E1 -1015.286,E2 -1015.286} C_VEL
LIN {X 0,Y 594.354,Z 467.608,A -85,B 0,C 180,E1 -1016.017,E2 -1016.017} C_VEL
LIN {X 0,Y 594.297,Z 474.397,A -85,B 0,C 180,E1 -1016.701,E2 -1016.701} C_VEL
LIN {X 0,Y 594.33,Z 480.933,A -85,B 0,C 180,E1 -1017.517,E2 -1017.517} C_VEL
LIN {X 0,Y 594.297,Z 485.619,A -85,B 0,C 180,E1 -1018.229,E2 -1018.229} C_VEL
LIN {X 0,Y 594.249,Z 489.766,A -85,B 0,C 180,E1 -1019.003,E2 -1019.003} C_VEL
LIN {X 0,Y 594.273,Z 493.063,A -85,B 0,C 180,E1 -1019.779,E2 -1019.779} C_VEL
LIN {X 0,Y 594.277,Z 495.607,A -85,B 0,C 180,E1 -1020.563,E2 -1020.563} C_VEL
LIN {X 0,Y 594.235,Z 497.843,A -85,B 0,C 180,E1 -1021.621,E2 -1021.621} C_VEL
LIN {X 0,Y 594.226,Z 498.568,A -85,B 0,C 180,E1 -1022.153,E2 -1022.153} C_VEL
LIN {X 0,Y 594.241,Z 498.983,A -85,B 0,C 180,E1 -1022.956,E2 -1022.956} C_VEL
LIN {X 0,Y 594.238,Z 498.329,A -85,B 0,C 180,E1 -1024.118,E2 -1024.118} C_VEL
LIN {X 0,Y 594.231,Z 497.675,A -85,B 0,C 180,E1 -1024.587,E2 -1024.587} C_VEL
LIN {X 0,Y 594.256,Z 494.696,A -85,B 0,C 180,E1 -1025.829,E2 -1025.829} C_VEL
LIN {X 0,Y 594.274,Z 491.251,A -85,B 0,C 180,E1 -1026.754,E2 -1026.754} C_VEL
LIN {X 0,Y 594.254,Z 487.139,A -85,B 0,C 180,E1 -1027.592,E2 -1027.592} C_VEL
LIN {X 0,Y 594.281,Z 482.692,A -85,B 0,C 180,E1 -1028.32,E2 -1028.32} C_VEL
LIN {X 0,Y 594.316,Z 477.461,A -85,B 0,C 180,E1 -1029.025,E2 -1029.025} C_VEL
LIN {X 0,Y 594.338,Z 470.725,A -85,B 0,C 180,E1 -1029.77,E2 -1029.77} C_VEL
LIN {X 0,Y 594.331,Z 461.812,A -85,B 0,C 180,E1 -1030.567,E2 -1030.567} C_VEL
LIN {X 0,Y 594.36,Z 452.729,A -85,B 0,C 180,E1 -1031.199,E2 -1031.199} C_VEL
LIN {X 0,Y 594.434,Z 443.01,A -85,B 0,C 180,E1 -1031.727,E2 -1031.727} C_VEL
LIN {X 0,Y 594.471,Z 433.32,A -85,B 0,C 180,E1 -1032.128,E2 -1032.128} C_VEL
LIN {X 0,Y 594.498,Z 424.123,A -85,B 0,C 180,E1 -1032.408,E2 -1032.408} C_VEL
LIN {X 0,Y 594.22,Z 419.38,A -85,B 0,C 180,E1 -1032.527,E2 -1032.527} C_VEL
LIN {X 0,Y 594.251,Z 412.873,A -85,B 0,C 180,E1 -1035.199,E2 -1035.199} C_VEL
LIN {X 0,Y 594.258,Z 407.051,A -85,B 0,C 180,E1 -1037.615,E2 -1037.615} C_VEL
LIN {X 0,Y 594.254,Z 400.635,A -85,B 0,C 180,E1 -1040.31,E2 -1040.31} C_VEL
LIN {X 0,Y 594.239,Z 394.55,A -85,B 0,C 180,E1 -1042.903,E2 -1042.903} C_VEL
LIN {X 0,Y 594.296,Z 387.705,A -85,B 0,C 180,E1 -1045.869,E2 -1045.869} C_VEL
LIN {X 0,Y 594.298,Z 381.434,A -85,B 0,C 180,E1 -1048.646,E2 -1048.646} C_VEL
LIN {X 0,Y 594.353,Z 374.638,A -85,B 0,C 180,E1 -1051.772,E2 -1051.772} C_VEL
LIN {X 0,Y 594.371,Z 369.615,A -85,B 0,C 180,E1 -1054.056,E2 -1054.056} C_VEL
LIN {X 0,Y 594.374,Z 366.449,A -85,B 0,C 180,E1 -1055.563,E2 -1055.563} C_VEL
LIN {X 0,Y 594.367,Z 366.451,A -85,B 0,C 180,E1 -1057.767,E2 -1057.767} C_VEL
LIN {X 0,Y 594.361,Z 366.449,A -85,B 0,C 180,E1 -1059.946,E2 -1059.946} C_VEL
LIN {X 0,Y 594.368,Z 366.451,A -85,B 0,C 180,E1 -1062.096,E2 -1062.096} C_VEL
LIN {X 0,Y 594.355,Z 366.451,A -85,B 0,C 180,E1 -1064.219,E2 -1064.219} C_VEL
LIN {X 0,Y 594.372,Z 366.448,A -85,B 0,C 180,E1 -1066.321,E2 -1066.321} C_VEL
LIN {X 0,Y 594.396,Z 366.445,A -85,B 0,C 180,E1 -1069.095,E2 -1069.095} C_VEL
LIN {X 0,Y 594.396,Z 366.444,A -85,B 0,C 180,E1 -1071.843,E2 -1071.843} C_VEL
LIN {X 0,Y 594.388,Z 366.445,A -85,B 0,C 180,E1 -1074.572,E2 -1074.572} C_VEL
LIN {X 0,Y 594.4,Z 366.444,A -85,B 0,C 180,E1 -1077.289,E2 -1077.289} C_VEL
LIN {X 0,Y 594.387,Z 366.446,A -85,B 0,C 180,E1 -1080,E2 -1080} C_VEL
LIN {X 0,Y 594.398,Z 366.444,A -85,B 0,C 180,E1 -1082.711,E2 -1082.711} C_VEL
LIN {X 0,Y 594.39,Z 366.445,A -85,B 0,C 180,E1 -1085.428,E2 -1085.428} C_VEL
LIN {X 0,Y 594.397,Z 366.445,A -85,B 0,C 180,E1 -1088.157,E2 -1088.157} C_VEL
LIN {X 0,Y 594.434,Z 366.442,A -85,B 0,C 180,E1 -1091.11,E2 -1091.11} C_VEL
LIN {X 0,Y 594.387,Z 366.446,A -85,B 0,C 180,E1 -1094.377,E2 -1094.377} C_VEL
LIN {X 0,Y 594.376,Z 366.447,A -85,B 0,C 180,E1 -1097.194,E2 -1097.194} C_VEL
LIN {X 0,Y 594.362,Z 366.449,A -85,B 0,C 180,E1 -1100.054,E2 -1100.054} C_VEL
LIN {X 0,Y 594.38,Z 366.447,A -85,B 0,C 180,E1 -1102.967,E2 -1102.967} C_VEL
LIN {X 0,Y 594.355,Z 366.45,A -85,B 0,C 180,E1 -1105.194,E2 -1105.194} C_VEL
LIN {X 0,Y 594.363,Z 366.451,A -85,B 0,C 180,E1 -1107.528,E2 -1107.528} C_VEL
LIN {X 0,Y 594.383,Z 366.447,A -85,B 0,C 180,E1 -1110.333,E2 -1110.333} C_VEL
LIN {X 0,Y 594.36,Z 366.451,A -85,B 0,C 180,E1 -1112.952,E2 -1112.952} C_VEL
LIN {X 0,Y 594.369,Z 366.452,A -85,B 0,C 180,E1 -1115.408,E2 -1115.408} C_VEL
LIN {X 0,Y 594.378,Z 366.45,A -85,B 0,C 180,E1 -1117.942,E2 -1117.942} C_VEL
LIN {X 0,Y 594.37,Z 366.451,A -85,B 0,C 180,E1 -1120.825,E2 -1120.825} C_VEL
LIN {X 0,Y 594.372,Z 366.451,A -85,B 0,C 180,E1 -1123.299,E2 -1123.299} C_VEL
LIN {X 0,Y 594.369,Z 366.451,A -85,B 0,C 180,E1 -1126.161,E2 -1126.161} C_VEL
LIN {X 0,Y 594.369,Z 366.448,A -85,B 0,C 180,E1 -1129.179,E2 -1129.179} C_VEL
LIN {X 0,Y 594.377,Z 366.447,A -85,B 0,C 180,E1 -1132.062,E2 -1132.062} C_VEL
LIN {X 0,Y 594.378,Z 366.447,A -85,B 0,C 180,E1 -1134.673,E2 -1134.673} C_VEL
LIN {X 0,Y 594.368,Z 366.45,A -85,B 0,C 180,E1 -1137.091,E2 -1137.091} C_VEL
LIN {X 0,Y 594.407,Z 366.536,A -85,B 0,C 180,E1 -1139.771,E2 -1139.771} C_VEL
LIN {X 0,Y 594.685,Z 370.278,A -85,B 0,C 180,E1 -1140.671,E2 -1140.671} C_VEL
LIN {X 0,Y 594.57,Z 381.847,A -85,B 0,C 180,E1 -1143.312,E2 -1143.312} C_VEL
LIN {X 0,Y 594.547,Z 393.623,A -85,B 0,C 180,E1 -1145.935,E2 -1145.935} C_VEL
LIN {X 0,Y 594.447,Z 406.933,A -85,B 0,C 180,E1 -1148.833,E2 -1148.833} C_VEL
LIN {X 0,Y 594.439,Z 418.857,A -85,B 0,C 180,E1 -1151.386,E2 -1151.386} C_VEL
LIN {X 0,Y 594.396,Z 430.633,A -85,B 0,C 180,E1 -1153.87,E2 -1153.87} C_VEL
LIN {X 0,Y 594.365,Z 444.091,A -85,B 0,C 180,E1 -1156.671,E2 -1156.671} C_VEL
LIN {X 0,Y 594.336,Z 450.085,A -85,B 0,C 180,E1 -1157.907,E2 -1157.907} C_VEL
LIN {X 0,Y 594.664,Z 455.043,A -85,B 0,C 180,E1 -1158.001,E2 -1158.001} C_VEL
LIN {X 0,Y 594.62,Z 468.279,A -85,B 0,C 180,E1 -1158.303,E2 -1158.303} C_VEL
LIN {X 0,Y 594.553,Z 480.469,A -85,B 0,C 180,E1 -1158.714,E2 -1158.714} C_VEL
LIN {X 0,Y 594.492,Z 492.666,A -85,B 0,C 180,E1 -1159.271,E2 -1159.271} C_VEL
LIN {X 0,Y 594.476,Z 504.226,A -85,B 0,C 180,E1 -1159.959,E2 -1159.959} C_VEL
LIN {X 0,Y 594.414,Z 514.617,A -85,B 0,C 180,E1 -1160.731,E2 -1160.731} C_VEL
LIN {X 0,Y 594.382,Z 523.13,A -85,B 0,C 180,E1 -1161.502,E2 -1161.502} C_VEL
LIN {X 0,Y 594.346,Z 530.975,A -85,B 0,C 180,E1 -1162.357,E2 -1162.357} C_VEL
LIN {X 0,Y 594.281,Z 538.82,A -85,B 0,C 180,E1 -1163.409,E2 -1163.409} C_VEL
LIN {X 0,Y 594.289,Z 545.689,A -85,B 0,C 180,E1 -1164.573,E2 -1164.573} C_VEL
LIN {X 0,Y 594.27,Z 550.378,A -85,B 0,C 180,E1 -1165.593,E2 -1165.593} C_VEL
LIN {X 0,Y 594.267,Z 553.962,A -85,B 0,C 180,E1 -1166.612,E2 -1166.612} C_VEL
LIN {X 0,Y 594.226,Z 555.813,A -85,B 0,C 180,E1 -1167.29,E2 -1167.29} C_VEL
LIN {X 0,Y 594.242,Z 557.204,A -85,B 0,C 180,E1 -1167.968,E2 -1167.968} C_VEL
LIN {X 0,Y 594.239,Z 558.785,A -85,B 0,C 180,E1 -1169.324,E2 -1169.324} C_VEL
LIN {X 0,Y 594.236,Z 559,A -85,B 0,C 180,E1 -1170.002,E2 -1170.002} C_VEL
LIN {X 0,Y 594.247,Z 558.183,A -85,B 0,C 180,E1 -1171.357,E2 -1171.357} C_VEL
LIN {X 0,Y 594.242,Z 557.199,A -85,B 0,C 180,E1 -1172.035,E2 -1172.035} C_VEL
LIN {X 0,Y 594.226,Z 555.805,A -85,B 0,C 180,E1 -1172.713,E2 -1172.713} C_VEL
LIN {X 0,Y 594.289,Z 552.891,A -85,B 0,C 180,E1 -1173.731,E2 -1173.731} C_VEL
LIN {X 0,Y 594.241,Z 548.944,A -85,B 0,C 180,E1 -1174.75,E2 -1174.75} C_VEL
LIN {X 0,Y 594.304,Z 542.869,A -85,B 0,C 180,E1 -1175.941,E2 -1175.941} C_VEL
LIN {X 0,Y 594.309,Z 536.226,A -85,B 0,C 180,E1 -1176.963,E2 -1176.963} C_VEL
LIN {X 0,Y 594.36,Z 527.978,A -85,B 0,C 180,E1 -1177.988,E2 -1177.988} C_VEL
LIN {X 0,Y 594.382,Z 519.522,A -85,B 0,C 180,E1 -1178.843,E2 -1178.843} C_VEL
LIN {X 0,Y 594.435,Z 509.076,A -85,B 0,C 180,E1 -1179.701,E2 -1179.701} C_VEL
LIN {X 0,Y 594.465,Z 498.737,A -85,B 0,C 180,E1 -1180.388,E2 -1180.388} C_VEL
LIN {X 0,Y 594.508,Z 486.693,A -85,B 0,C 180,E1 -1181.022,E2 -1181.022} C_VEL
LIN {X 0,Y 594.566,Z 474.45,A -85,B 0,C 180,E1 -1181.507,E2 -1181.507} C_VEL
LIN {X 0,Y 594.647,Z 461.387,A -85,B 0,C 180,E1 -1181.873,E2 -1181.873} C_VEL
LIN {X 0,Y 594.52,Z 451.457,A -85,B 0,C 180,E1 -1182.057,E2 -1182.057} C_VEL
LIN {X 0,Y 594.334,Z 450.07,A -85,B 0,C 180,E1 -1182.096,E2 -1182.096} C_VEL
LIN {X 0,Y 594.343,Z 437.347,A -85,B 0,C 180,E1 -1184.729,E2 -1184.729} C_VEL
LIN {X 0,Y 594.408,Z 425.571,A -85,B 0,C 180,E1 -1187.194,E2 -1187.194} C_VEL
LIN {X 0,Y 594.464,Z 412.113,A -85,B 0,C 180,E1 -1190.052,E2 -1190.052} C_VEL
LIN {X 0,Y 594.482,Z 398.655,A -85,B 0,C 180,E1 -1192.964,E2 -1192.964} C_VEL
LIN {X 0,Y 594.564,Z 386.879,A -85,B 0,C 180,E1 -1195.56,E2 -1195.56} C_VEL
LIN {X 0,Y 594.641,Z 375.103,A -85,B 0,C 180,E1 -1198.214,E2 -1198.214} C_VEL
LIN {X 0,Y 594.653,Z 368.351,A -85,B 0,C 180,E1 -1199.762,E2 -1199.762} C_VEL
LIN {X 0,Y 594.367,Z 366.449,A -85,B 0,C 180,E1 -1200.26,E2 -1200.26} C_VEL
LIN {X 0,Y 594.381,Z 366.45,A -85,B 0,C 180,E1 -1202.951,E2 -1202.951} C_VEL
LIN {X 0,Y 594.357,Z 366.446,A -85,B 0,C 180,E1 -1205.409,E2 -1205.409} C_VEL
LIN {X 0,Y 594.388,Z 366.446,A -85,B 0,C 180,E1 -1207.941,E2 -1207.941} C_VEL
LIN {X 0,Y 594.365,Z 366.444,A -85,B 0,C 180,E1 -1210.82,E2 -1210.82} C_VEL
LIN {X 0,Y 594.337,Z 366.452,A -85,B 0,C 180,E1 -1213.836,E2 -1213.836} C_VEL
LIN {X 0,Y 594.347,Z 366.448,A -85,B 0,C 180,E1 -1216.698,E2 -1216.698} C_VEL
LIN {X 0,Y 594.366,Z 366.446,A -85,B 0,C 180,E1 -1219.432,E2 -1219.432} C_VEL
LIN {X 0,Y 594.391,Z 366.447,A -85,B 0,C 180,E1 -1222.392,E2 -1222.392} C_VEL
LIN {X 0,Y 594.38,Z 366.443,A -85,B 0,C 180,E1 -1225.42,E2 -1225.42} C_VEL
LIN {X 0,Y 594.376,Z 366.445,A -85,B 0,C 180,E1 -1228.358,E2 -1228.358} C_VEL
LIN {X 0,Y 594.38,Z 366.444,A -85,B 0,C 180,E1 -1231.043,E2 -1231.043} C_VEL
LIN {X 0,Y 594.341,Z 366.447,A -85,B 0,C 180,E1 -1234.054,E2 -1234.054} C_VEL
LIN {X 0,Y 594.355,Z 366.452,A -85,B 0,C 180,E1 -1237.032,E2 -1237.032} C_VEL
LIN {X 0,Y 594.368,Z 366.446,A -85,B 0,C 180,E1 -1239.946,E2 -1239.946} C_VEL
LIN {X 0,Y 594.39,Z 366.443,A -85,B 0,C 180,E1 -1242.806,E2 -1242.806} C_VEL
LIN {X 0,Y 594.391,Z 366.45,A -85,B 0,C 180,E1 -1245.827,E2 -1245.827} C_VEL
LIN {X 0,Y 594.393,Z 366.443,A -85,B 0,C 180,E1 -1248.926,E2 -1248.926} C_VEL
LIN {X 0,Y 594.339,Z 366.449,A -85,B 0,C 180,E1 -1251.842,E2 -1251.842} C_VEL
LIN {X 0,Y 594.382,Z 366.447,A -85,B 0,C 180,E1 -1254.572,E2 -1254.572} C_VEL
LIN {X 0,Y 594.322,Z 366.576,A -85,B 0,C 180,E1 -1256.568,E2 -1256.568} C_VEL
LIN {X 0,Y 594.311,Z 372.266,A -85,B 0,C 180,E1 -1258.645,E2 -1258.645} C_VEL
LIN {X 0,Y 594.363,Z 377.739,A -85,B 0,C 180,E1 -1260.677,E2 -1260.677} C_VEL
LIN {X 0,Y 594.402,Z 382.875,A -85,B 0,C 180,E1 -1262.711,E2 -1262.711} C_VEL
LIN {X 0,Y 594.358,Z 389.33,A -85,B 0,C 180,E1 -1265.428,E2 -1265.428} C_VEL
LIN {X 0,Y 594.34,Z 395.96,A -85,B 0,C 180,E1 -1268.157,E2 -1268.157} C_VEL
LIN {X 0,Y 594.312,Z 403.093,A -85,B 0,C 180,E1 -1271.034,E2 -1271.034} C_VEL
LIN {X 0,Y 594.28,Z 410.916,A -85,B 0,C 180,E1 -1274.131,E2 -1274.131} C_VEL
LIN {X 0,Y 594.27,Z 413.206,A -85,B 0,C 180,E1 -1275.027,E2 -1275.027} C_VEL
LIN {X 0,Y 593.608,Z 414.657,A -85,B 0,C 180,E1 -1275.576,E2 -1275.576} C_VEL
LIN {X 0,Y 590.709,Z 417.121,A -85,B 0,C 180,E1 -1276.462,E2 -1276.462} C_VEL
LIN {X 0,Y 588.256,Z 419.101,A -85,B 0,C 180,E1 -1277.174,E2 -1277.174} C_VEL
LIN {X 0,Y 587.212,Z 420.576,A -85,B 0,C 180,E1 -1277.726,E2 -1277.726} C_VEL
LIN {X 0,Y 587.132,Z 421.06,A -85,B 0,C 180,E1 -1277.913,E2 -1277.913} C_VEL
LIN {X 0,Y 587.201,Z 423.593,A -85,B 0,C 180,E1 -1278.869,E2 -1278.869} C_VEL
LIN {X 0,Y 587.733,Z 429.571,A -85,B 0,C 180,E1 -1278.989,E2 -1278.989} C_VEL
LIN {X 0,Y 587.651,Z 441.847,A -85,B 0,C 180,E1 -1279.315,E2 -1279.315} C_VEL
LIN {X 0,Y 587.557,Z 453.445,A -85,B 0,C 180,E1 -1279.749,E2 -1279.749} C_VEL
LIN {X 0,Y 587.501,Z 464.693,A -85,B 0,C 180,E1 -1280.298,E2 -1280.298} C_VEL
LIN {X 0,Y 587.453,Z 476.407,A -85,B 0,C 180,E1 -1281.033,E2 -1281.033} C_VEL
LIN {X 0,Y 587.364,Z 486.953,A -85,B 0,C 180,E1 -1281.865,E2 -1281.865} C_VEL
LIN {X 0,Y 587.294,Z 495.516,A -85,B 0,C 180,E1 -1282.693,E2 -1282.693} C_VEL
LIN {X 0,Y 587.258,Z 503.538,A -85,B 0,C 180,E1 -1283.635,E2 -1283.635} C_VEL
LIN {X 0,Y 587.227,Z 511.292,A -85,B 0,C 180,E1 -1284.764,E2 -1284.764} C_VEL
LIN {X 0,Y 587.187,Z 517.108,A -85,B 0,C 180,E1 -1285.838,E2 -1285.838} C_VEL
LIN {X 0,Y 587.144,Z 522.146,A -85,B 0,C 180,E1 -1287.055,E2 -1287.055} C_VEL
LIN {X 0,Y 587.175,Z 524.588,A -85,B 0,C 180,E1 -1287.826,E2 -1287.826} C_VEL
LIN {X 0,Y 587.166,Z 527.385,A -85,B 0,C 180,E1 -1289.101,E2 -1289.101} C_VEL
LIN {X 0,Y 587.155,Z 528.863,A -85,B 0,C 180,E1 -1290.479,E2 -1290.479} C_VEL
LIN {X 0,Y 587.133,Z 528.736,A -85,B 0,C 180,E1 -1291.802,E2 -1291.802} C_VEL
LIN {X 0,Y 587.144,Z 527.234,A -85,B 0,C 180,E1 -1293.082,E2 -1293.082} C_VEL
LIN {X 0,Y 587.159,Z 524.432,A -85,B 0,C 180,E1 -1294.32,E2 -1294.32} C_VEL
LIN {X 0,Y 587.169,Z 520.323,A -85,B 0,C 180,E1 -1295.519,E2 -1295.519} C_VEL
LIN {X 0,Y 587.228,Z 514.547,A -85,B 0,C 180,E1 -1296.755,E2 -1296.755} C_VEL
LIN {X 0,Y 587.205,Z 508.14,A -85,B 0,C 180,E1 -1297.821,E2 -1297.821} C_VEL
LIN {X 0,Y 587.268,Z 501.542,A -85,B 0,C 180,E1 -1298.711,E2 -1298.711} C_VEL
LIN {X 0,Y 587.319,Z 492.635,A -85,B 0,C 180,E1 -1299.694,E2 -1299.694} C_VEL
LIN {X 0,Y 587.383,Z 482.664,A -85,B 0,C 180,E1 -1300.586,E2 -1300.586} C_VEL
LIN {X 0,Y 587.437,Z 471.687,A -85,B 0,C 180,E1 -1301.376,E2 -1301.376} C_VEL
LIN {X 0,Y 587.489,Z 459.578,A -85,B 0,C 180,E1 -1302.06,E2 -1302.06} C_VEL
LIN {X 0,Y 587.585,Z 447.139,A -85,B 0,C 180,E1 -1302.596,E2 -1302.596} C_VEL
LIN {X 0,Y 587.701,Z 433.873,A -85,B 0,C 180,E1 -1303.002,E2 -1303.002} C_VEL
LIN {X 0,Y 587.555,Z 426.156,A -85,B 0,C 180,E1 -1303.171,E2 -1303.171} C_VEL
LIN {X 0,Y 587.136,Z 423.457,A -85,B 0,C 180,E1 -1303.243,E2 -1303.243} C_VEL
LIN {X 0,Y 587.17,Z 416.317,A -85,B 0,C 180,E1 -1306.034,E2 -1306.034} C_VEL
LIN {X 0,Y 587.155,Z 408.973,A -85,B 0,C 180,E1 -1308.945,E2 -1308.945} C_VEL
LIN {X 0,Y 587.196,Z 402.597,A -85,B 0,C 180,E1 -1311.509,E2 -1311.509} C_VEL
LIN {X 0,Y 587.23,Z 395.366,A -85,B 0,C 180,E1 -1314.471,E2 -1314.471} C_VEL
LIN {X 0,Y 587.237,Z 389.549,A -85,B 0,C 180,E1 -1316.903,E2 -1316.903} C_VEL
LIN {X 0,Y 587.263,Z 384.436,A -85,B 0,C 180,E1 -1319.029,E2 -1319.029} C_VEL
LIN {X 0,Y 587.252,Z 378.63,A -85,B 0,C 180,E1 -1321.398,E2 -1321.398} C_VEL
LIN {X 0,Y 587.298,Z 372.634,A -85,B 0,C 180,E1 -1323.831,E2 -1323.831} C_VEL
LIN {X 0,Y 587.332,Z 367.326,A -85,B 0,C 180,E1 -1325.992,E2 -1325.992} C_VEL
LIN {X 0,Y 587.323,Z 367.324,A -85,B 0,C 180,E1 -1328.225,E2 -1328.225} C_VEL
LIN {X 0,Y 587.328,Z 367.323,A -85,B 0,C 180,E1 -1331.149,E2 -1331.149} C_VEL
LIN {X 0,Y 587.323,Z 367.325,A -85,B 0,C 180,E1 -1334.024,E2 -1334.024} C_VEL
LIN {X 0,Y 587.364,Z 367.319,A -85,B 0,C 180,E1 -1336.153,E2 -1336.153} C_VEL
LIN {X 0,Y 587.338,Z 367.322,A -85,B 0,C 180,E1 -1338.961,E2 -1338.961} C_VEL
LIN {X 0,Y 587.367,Z 367.321,A -85,B 0,C 180,E1 -1341.743,E2 -1341.743} C_VEL
LIN {X 0,Y 587.354,Z 367.326,A -85,B 0,C 180,E1 -1344.506,E2 -1344.506} C_VEL
LIN {X 0,Y 587.372,Z 367.321,A -85,B 0,C 180,E1 -1347.941,E2 -1347.941} C_VEL
LIN {X 0,Y 587.384,Z 367.434,A -85,B 0,C 180,E1 -1350.598,E2 -1350.598} C_VEL
LIN {X 0,Y 587.373,Z 372.025,A -85,B 0,C 180,E1 -1352.742,E2 -1352.742} C_VEL
LIN {X 0,Y 587.327,Z 377.918,A -85,B 0,C 180,E1 -1355.492,E2 -1355.492} C_VEL
LIN {X 0,Y 587.265,Z 383.954,A -85,B 0,C 180,E1 -1358.255,E2 -1358.255} C_VEL
LIN {X 0,Y 587.257,Z 390.319,A -85,B 0,C 180,E1 -1361.088,E2 -1361.088} C_VEL
LIN {X 0,Y 587.213,Z 397.464,A -85,B 0,C 180,E1 -1364.202,E2 -1364.202} C_VEL
LIN {X 0,Y 587.194,Z 403.442,A -85,B 0,C 180,E1 -1366.764,E2 -1366.764} C_VEL
LIN {X 0,Y 587.137,Z 410.103,A -85,B 0,C 180,E1 -1369.58,E2 -1369.58} C_VEL
LIN {X 0,Y 587.127,Z 415.36,A -85,B 0,C 180,E1 -1371.78,E2 -1371.78} C_VEL
LIN {X 0,Y 587.175,Z 419.427,A -85,B 0,C 180,E1 -1373.449,E2 -1373.449} C_VEL
LIN {X 0,Y 587.518,Z 426.97,A -85,B 0,C 180,E1 -1373.645,E2 -1373.645} C_VEL
LIN {X 0,Y 587.413,Z 439.284,A -85,B 0,C 180,E1 -1374.084,E2 -1374.084} C_VEL
LIN {X 0,Y 587.303,Z 448.968,A -85,B 0,C 180,E1 -1374.57,E2 -1374.57} C_VEL
LIN {X 0,Y 587.288,Z 457.825,A -85,B 0,C 180,E1 -1375.137,E2 -1375.137} C_VEL
LIN {X 0,Y 587.311,Z 466.151,A -85,B 0,C 180,E1 -1375.801,E2 -1375.801} C_VEL
LIN {X 0,Y 587.232,Z 474.742,A -85,B 0,C 180,E1 -1376.664,E2 -1376.664} C_VEL
LIN {X 0,Y 587.258,Z 480.805,A -85,B 0,C 180,E1 -1377.43,E2 -1377.43} C_VEL
LIN {X 0,Y 587.205,Z 486.936,A -85,B 0,C 180,E1 -1378.406,E2 -1378.406} C_VEL
LIN {X 0,Y 587.188,Z 491.674,A -85,B 0,C 180,E1 -1379.386,E2 -1379.386} C_VEL
LIN {X 0,Y 587.176,Z 495.477,A -85,B 0,C 180,E1 -1380.484,E2 -1380.484} C_VEL
LIN {X 0,Y 587.133,Z 498.086,A -85,B 0,C 180,E1 -1381.779,E2 -1381.779} C_VEL
LIN {X 0,Y 587.134,Z 498.997,A -85,B 0,C 180,E1 -1383.081,E2 -1383.081} C_VEL
LIN {X 0,Y 587.131,Z 498.078,A -85,B 0,C 180,E1 -1384.317,E2 -1384.317} C_VEL
LIN {X 0,Y 587.141,Z 495.704,A -85,B 0,C 180,E1 -1385.517,E2 -1385.517} C_VEL
LIN {X 0,Y 587.203,Z 491.742,A -85,B 0,C 180,E1 -1386.689,E2 -1386.689} C_VEL
LIN {X 0,Y 587.173,Z 487.309,A -85,B 0,C 180,E1 -1387.618,E2 -1387.618} C_VEL
LIN {X 0,Y 587.209,Z 482,A -85,B 0,C 180,E1 -1388.486,E2 -1388.486} C_VEL
LIN {X 0,Y 587.254,Z 475.273,A -85,B 0,C 180,E1 -1389.364,E2 -1389.364} C_VEL
LIN {X 0,Y 587.315,Z 466.579,A -85,B 0,C 180,E1 -1390.251,E2 -1390.251} C_VEL
LIN {X 0,Y 587.329,Z 458.788,A -85,B 0,C 180,E1 -1390.884,E2 -1390.884} C_VEL
LIN {X 0,Y 587.339,Z 451.339,A -85,B 0,C 180,E1 -1391.381,E2 -1391.381} C_VEL
LIN {X 0,Y 587.43,Z 443.002,A -85,B 0,C 180,E1 -1391.832,E2 -1391.832} C_VEL
LIN {X 0,Y 587.475,Z 434.179,A -85,B 0,C 180,E1 -1392.207,E2 -1392.207} C_VEL
LIN {X 0,Y 587.501,Z 424.157,A -85,B 0,C 180,E1 -1392.52,E2 -1392.52} C_VEL
LIN {X 0,Y 587.168,Z 419.323,A -85,B 0,C 180,E1 -1392.662,E2 -1392.662} C_VEL
LIN {X 0,Y 587.164,Z 413.527,A -85,B 0,C 180,E1 -1395.074,E2 -1395.074} C_VEL
LIN {X 0,Y 587.172,Z 406.775,A -85,B 0,C 180,E1 -1397.912,E2 -1397.912} C_VEL
LIN {X 0,Y 587.165,Z 400.398,A -85,B 0,C 180,E1 -1400.627,E2 -1400.627} C_VEL
LIN {X 0,Y 587.186,Z 394.188,A -85,B 0,C 180,E1 -1403.309,E2 -1403.309} C_VEL
LIN {X 0,Y 587.241,Z 388.576,A -85,B 0,C 180,E1 -1405.772,E2 -1405.772} C_VEL
LIN {X 0,Y 587.231,Z 383.093,A -85,B 0,C 180,E1 -1408.225,E2 -1408.225} C_VEL
LIN {X 0,Y 587.299,Z 377.412,A -85,B 0,C 180,E1 -1410.87,E2 -1410.87} C_VEL
LIN {X 0,Y 587.345,Z 371.004,A -85,B 0,C 180,E1 -1413.816,E2 -1413.816} C_VEL
LIN {X 0,Y 587.337,Z 367.326,A -85,B 0,C 180,E1 -1415.596,E2 -1415.596} C_VEL
LIN {X 0,Y 587.315,Z 367.328,A -85,B 0,C 180,E1 -1418.226,E2 -1418.226} C_VEL
LIN {X 0,Y 587.348,Z 367.323,A -85,B 0,C 180,E1 -1421.151,E2 -1421.151} C_VEL
LIN {X 0,Y 587.311,Z 367.328,A -85,B 0,C 180,E1 -1424.025,E2 -1424.025} C_VEL
LIN {X 0,Y 587.356,Z 367.324,A -85,B 0,C 180,E1 -1426.154,E2 -1426.154} C_VEL
LIN {X 0,Y 587.386,Z 367.319,A -85,B 0,C 180,E1 -1428.964,E2 -1428.964} C_VEL
LIN {X 0,Y 587.35,Z 367.323,A -85,B 0,C 180,E1 -1431.745,E2 -1431.745} C_VEL
LIN {X 0,Y 587.354,Z 367.322,A -85,B 0,C 180,E1 -1434.507,E2 -1434.507} C_VEL
LIN {X 0,Y 587.365,Z 367.32,A -85,B 0,C 180,E1 -1437.257,E2 -1437.257} C_VEL
LIN {X 0,Y 587.356,Z 367.321,A -85,B 0,C 180,E1 -1440,E2 -1440} C_VEL
LIN {X 0,Y 587.363,Z 367.321,A -85,B 0,C 180,E1 -1442.744,E2 -1442.744} C_VEL
LIN {X 0,Y 587.355,Z 367.322,A -85,B 0,C 180,E1 -1445.493,E2 -1445.493} C_VEL
LIN {X 0,Y 587.351,Z 367.323,A -85,B 0,C 180,E1 -1448.256,E2 -1448.256} C_VEL
LIN {X 0,Y 587.405,Z 367.318,A -85,B 0,C 180,E1 -1451.176,E2 -1451.176} C_VEL
LIN {X 0,Y 587.329,Z 367.325,A -85,B 0,C 180,E1 -1454.554,E2 -1454.554} C_VEL
LIN {X 0,Y 587.343,Z 367.323,A -85,B 0,C 180,E1 -1457.406,E2 -1457.406} C_VEL
LIN {X 0,Y 587.317,Z 367.327,A -85,B 0,C 180,E1 -1460.306,E2 -1460.306} C_VEL
LIN {X 0,Y 587.346,Z 367.326,A -85,B 0,C 180,E1 -1463.258,E2 -1463.258} C_VEL
LIN {X 0,Y 587.344,Z 367.324,A -85,B 0,C 180,E1 -1466.279,E2 -1466.279} C_VEL
LIN {X 0,Y 587.335,Z 367.324,A -85,B 0,C 180,E1 -1469.136,E2 -1469.136} C_VEL
LIN {X 0,Y 587.34,Z 367.323,A -85,B 0,C 180,E1 -1471.84,E2 -1471.84} C_VEL
LIN {X 0,Y 587.345,Z 367.324,A -85,B 0,C 180,E1 -1474.352,E2 -1474.352} C_VEL
LIN {X 0,Y 587.335,Z 367.328,A -85,B 0,C 180,E1 -1476.748,E2 -1476.748} C_VEL
LIN {X 0,Y 587.333,Z 367.329,A -85,B 0,C 180,E1 -1479.361,E2 -1479.361} C_VEL
LIN {X 0,Y 587.351,Z 367.326,A -85,B 0,C 180,E1 -1482.113,E2 -1482.113} C_VEL
LIN {X 0,Y 587.301,Z 367.329,A -85,B 0,C 180,E1 -1485.091,E2 -1485.091} C_VEL
LIN {X 0,Y 587.339,Z 367.324,A -85,B 0,C 180,E1 -1487.93,E2 -1487.93} C_VEL
LIN {X 0,Y 587.325,Z 367.327,A -85,B 0,C 180,E1 -1491.06,E2 -1491.06} C_VEL
LIN {X 0,Y 587.343,Z 367.324,A -85,B 0,C 180,E1 -1493.294,E2 -1493.294} C_VEL
LIN {X 0,Y 587.362,Z 367.322,A -85,B 0,C 180,E1 -1495.783,E2 -1495.783} C_VEL
LIN {X 0,Y 587.342,Z 367.327,A -85,B 0,C 180,E1 -1498.234,E2 -1498.234} C_VEL
LIN {X 0,Y 587.387,Z 367.51,A -85,B 0,C 180,E1 -1499.586,E2 -1499.586} C_VEL
LIN {X 0,Y 587.758,Z 371.873,A -85,B 0,C 180,E1 -1500.646,E2 -1500.646} C_VEL
LIN {X 0,Y 587.631,Z 383.529,A -85,B 0,C 180,E1 -1503.355,E2 -1503.355} C_VEL
LIN {X 0,Y 587.571,Z 395.305,A -85,B 0,C 180,E1 -1506.006,E2 -1506.006} C_VEL
LIN {X 0,Y 587.443,Z 407.083,A -85,B 0,C 180,E1 -1508.602,E2 -1508.602} C_VEL
LIN {X 0,Y 587.414,Z 418.857,A -85,B 0,C 180,E1 -1511.155,E2 -1511.155} C_VEL
LIN {X 0,Y 587.367,Z 430.633,A -85,B 0,C 180,E1 -1513.671,E2 -1513.671} C_VEL
LIN {X 0,Y 587.31,Z 444.091,A -85,B 0,C 180,E1 -1516.508,E2 -1516.508} C_VEL
LIN {X 0,Y 587.269,Z 450.085,A -85,B 0,C 180,E1 -1517.76,E2 -1517.76} C_VEL
LIN {X 0,Y 587.725,Z 455.043,A -85,B 0,C 180,E1 -1517.857,E2 -1517.857} C_VEL
LIN {X 0,Y 587.688,Z 468.279,A -85,B 0,C 180,E1 -1518.163,E2 -1518.163} C_VEL
LIN {X 0,Y 587.582,Z 481.003,A -85,B 0,C 180,E1 -1518.599,E2 -1518.599} C_VEL
LIN {X 0,Y 587.513,Z 492.665,A -85,B 0,C 180,E1 -1519.142,E2 -1519.142} C_VEL
LIN {X 0,Y 587.472,Z 504.227,A -85,B 0,C 180,E1 -1519.838,E2 -1519.838} C_VEL
LIN {X 0,Y 587.366,Z 514.619,A -85,B 0,C 180,E1 -1520.619,E2 -1520.619} C_VEL
LIN {X 0,Y 587.321,Z 523.13,A -85,B 0,C 180,E1 -1521.399,E2 -1521.399} C_VEL
LIN {X 0,Y 587.273,Z 530.975,A -85,B 0,C 180,E1 -1522.264,E2 -1522.264} C_VEL
LIN {X 0,Y 587.231,Z 537.482,A -85,B 0,C 180,E1 -1523.128,E2 -1523.128} C_VEL
LIN {X 0,Y 587.236,Z 543.875,A -85,B 0,C 180,E1 -1524.163,E2 -1524.163} C_VEL
LIN {X 0,Y 587.147,Z 548.956,A -85,B 0,C 180,E1 -1525.195,E2 -1525.195} C_VEL
LIN {X 0,Y 587.213,Z 552.901,A -85,B 0,C 180,E1 -1526.227,E2 -1526.227} C_VEL
LIN {X 0,Y 587.132,Z 555.813,A -85,B 0,C 180,E1 -1527.257,E2 -1527.257} C_VEL
LIN {X 0,Y 587.141,Z 557.204,A -85,B 0,C 180,E1 -1527.944,E2 -1527.944} C_VEL
LIN {X 0,Y 587.14,Z 558.785,A -85,B 0,C 180,E1 -1529.316,E2 -1529.316} C_VEL
LIN {X 0,Y 587.137,Z 559,A -85,B 0,C 180,E1 -1530.002,E2 -1530.002} C_VEL
LIN {X 0,Y 587.147,Z 558.183,A -85,B 0,C 180,E1 -1531.373,E2 -1531.373} C_VEL
LIN {X 0,Y 587.141,Z 557.198,A -85,B 0,C 180,E1 -1532.059,E2 -1532.059} C_VEL
LIN {X 0,Y 587.132,Z 555.805,A -85,B 0,C 180,E1 -1532.746,E2 -1532.746} C_VEL
LIN {X 0,Y 587.213,Z 552.891,A -85,B 0,C 180,E1 -1533.776,E2 -1533.776} C_VEL
LIN {X 0,Y 587.147,Z 548.944,A -85,B 0,C 180,E1 -1534.808,E2 -1534.808} C_VEL
LIN {X 0,Y 587.217,Z 542.869,A -85,B 0,C 180,E1 -1536.013,E2 -1536.013} C_VEL
LIN {X 0,Y 587.246,Z 536.227,A -85,B 0,C 180,E1 -1537.048,E2 -1537.048} C_VEL
LIN {X 0,Y 587.3,Z 527.978,A -85,B 0,C 180,E1 -1538.084,E2 -1538.084} C_VEL
LIN {X 0,Y 587.344,Z 519.523,A -85,B 0,C 180,E1 -1538.95,E2 -1538.95} C_VEL
LIN {X 0,Y 587.421,Z 509.078,A -85,B 0,C 180,E1 -1539.818,E2 -1539.818} C_VEL
LIN {X 0,Y 587.481,Z 498.737,A -85,B 0,C 180,E1 -1540.513,E2 -1540.513} C_VEL
LIN {X 0,Y 587.534,Z 487.116,A -85,B 0,C 180,E1 -1541.135,E2 -1541.135} C_VEL
LIN {X 0,Y 587.627,Z 474.649,A -85,B 0,C 180,E1 -1541.638,E2 -1541.638} C_VEL
LIN {X 0,Y 587.697,Z 461.386,A -85,B 0,C 180,E1 -1542.015,E2 -1542.015} C_VEL
LIN {X 0,Y 587.589,Z 452.211,A -85,B 0,C 180,E1 -1542.19,E2 -1542.19} C_VEL
LIN {X 0,Y 587.271,Z 450.07,A -85,B 0,C 180,E1 -1542.243,E2 -1542.243} C_VEL
LIN {X 0,Y 587.304,Z 437.347,A -85,B 0,C 180,E1 -1544.91,E2 -1544.91} C_VEL
LIN {X 0,Y 587.379,Z 425.571,A -85,B 0,C 180,E1 -1547.406,E2 -1547.406} C_VEL
LIN {X 0,Y 587.457,Z 412.113,A -85,B 0,C 180,E1 -1550.301,E2 -1550.301} C_VEL
LIN {X 0,Y 587.526,Z 398.655,A -85,B 0,C 180,E1 -1553.251,E2 -1553.251} C_VEL
LIN {X 0,Y 587.613,Z 386.955,A -85,B 0,C 180,E1 -1555.868,E2 -1555.868} C_VEL
LIN {X 0,Y 587.684,Z 375.046,A -85,B 0,C 180,E1 -1558.579,E2 -1558.579} C_VEL
LIN {X 0,Y 587.743,Z 370.076,A -85,B 0,C 180,E1 -1559.753,E2 -1559.753} C_VEL
LIN {X 0,Y 587.338,Z 367.326,A -85,B 0,C 180,E1 -1560.444,E2 -1560.444} C_VEL
LIN {X 0,Y 587.343,Z 367.324,A -85,B 0,C 180,E1 -1563.112,E2 -1563.112} C_VEL
LIN {X 0,Y 587.304,Z 367.325,A -85,B 0,C 180,E1 -1565.538,E2 -1565.538} C_VEL
LIN {X 0,Y 587.324,Z 367.326,A -85,B 0,C 180,E1 -1568.481,E2 -1568.481} C_VEL
LIN {X 0,Y 587.315,Z 367.323,A -85,B 0,C 180,E1 -1571.16,E2 -1571.16} C_VEL
LIN {X 0,Y 587.289,Z 367.327,A -85,B 0,C 180,E1 -1574.109,E2 -1574.109} C_VEL
LIN {X 0,Y 587.295,Z 367.33,A -85,B 0,C 180,E1 -1576.991,E2 -1576.991} C_VEL
LIN {X 0,Y 587.312,Z 367.323,A -85,B 0,C 180,E1 -1579.745,E2 -1579.745} C_VEL
LIN {X 0,Y 587.346,Z 367.324,A -85,B 0,C 180,E1 -1582.392,E2 -1582.392} C_VEL
LIN {X 0,Y 587.346,Z 367.321,A -85,B 0,C 180,E1 -1585.653,E2 -1585.653} C_VEL
LIN {X 0,Y 587.341,Z 367.323,A -85,B 0,C 180,E1 -1588.231,E2 -1588.231} C_VEL
LIN {X 0,Y 587.345,Z 367.32,A -85,B 0,C 180,E1 -1590.868,E2 -1590.868} C_VEL
LIN {X 0,Y 587.295,Z 367.326,A -85,B 0,C 180,E1 -1593.832,E2 -1593.832} C_VEL
LIN {X 0,Y 587.304,Z 367.33,A -85,B 0,C 180,E1 -1596.74,E2 -1596.74} C_VEL
LIN {X 0,Y 587.325,Z 367.322,A -85,B 0,C 180,E1 -1599.695,E2 -1599.695} C_VEL
LIN {X 0,Y 587.309,Z 367.326,A -85,B 0,C 180,E1 -1601.873,E2 -1601.873} C_VEL
LIN {X 0,Y 587.323,Z 367.33,A -85,B 0,C 180,E1 -1604.025,E2 -1604.025} C_VEL
LIN {X 0,Y 587.355,Z 367.322,A -85,B 0,C 180,E1 -1606.154,E2 -1606.154} C_VEL
LIN {X 0,Y 587.344,Z 367.321,A -85,B 0,C 180,E1 -1608.962,E2 -1608.962} C_VEL
LIN {X 0,Y 587.308,Z 367.325,A -85,B 0,C 180,E1 -1611.744,E2 -1611.744} C_VEL
LIN {X 0,Y 587.344,Z 367.323,A -85,B 0,C 180,E1 -1614.507,E2 -1614.507} C_VEL
LIN {X 0,Y 587.241,Z 367.472,A -85,B 0,C 180,E1 -1616.655,E2 -1616.655} C_VEL
LIN {X 0,Y 587.271,Z 374.705,A -85,B 0,C 180,E1 -1619.314,E2 -1619.314} C_VEL
LIN {X 0,Y 587.305,Z 380.126,A -85,B 0,C 180,E1 -1621.371,E2 -1621.371} C_VEL
LIN {X 0,Y 587.281,Z 387.023,A -85,B 0,C 180,E1 -1624.117,E2 -1624.117} C_VEL
LIN {X 0,Y 587.273,Z 393.025,A -85,B 0,C 180,E1 -1626.647,E2 -1626.647} C_VEL
LIN {X 0,Y 587.259,Z 398.594,A -85,B 0,C 180,E1 -1628.95,E2 -1628.95} C_VEL
LIN {X 0,Y 587.234,Z 403.816,A -85,B 0,C 180,E1 -1631.075,E2 -1631.075} C_VEL
LIN {X 0,Y 587.204,Z 411.612,A -85,B 0,C 180,E1 -1634.197,E2 -1634.197} C_VEL
LIN {X 0,Y 587.178,Z 418.104,A -85,B 0,C 180,E1 -1636.758,E2 -1636.758} C_VEL
LIN {X 0,Y 587.132,Z 421.06,A -85,B 0,C 180,E1 -1637.913,E2 -1637.913} C_VEL
LIN {X 0,Y 586.813,Z 422.659,A -85,B 0,C 180,E1 -1638.242,E2 -1638.242} C_VEL
LIN {X 0,Y 586.043,Z 425.19,A -85,B 0,C 180,E1 -1638.509,E2 -1638.509} C_VEL
LIN {X 0,Y 584.453,Z 430.004,A -85,B 0,C 180,E1 -1638.806,E2 -1638.806} C_VEL
LIN {X 0,Y 582.635,Z 435.679,A -85,B 0,C 180,E1 -1639.009,E2 -1639.009} C_VEL
LIN {X 0,Y 581.134,Z 441.792,A -85,B 0,C 180,E1 -1639.18,E2 -1639.18} C_VEL
LIN {X 0,Y 580.648,Z 447.855,A -85,B 0,C 180,E1 -1639.382,E2 -1639.382} C_VEL
LIN {X 0,Y 580.526,Z 461.596,A -85,B 0,C 180,E1 -1639.999,E2 -1639.999} C_VEL
LIN {X 0,Y 580.457,Z 472.446,A -85,B 0,C 180,E1 -1640.641,E2 -1640.641} C_VEL
LIN {X 0,Y 580.366,Z 482.728,A -85,B 0,C 180,E1 -1641.395,E2 -1641.395} C_VEL
LIN {X 0,Y 580.282,Z 492.117,A -85,B 0,C 180,E1 -1642.239,E2 -1642.239} C_VEL
LIN {X 0,Y 580.211,Z 501.205,A -85,B 0,C 180,E1 -1643.244,E2 -1643.244} C_VEL
LIN {X 0,Y 580.157,Z 508.996,A -85,B 0,C 180,E1 -1644.322,E2 -1644.322} C_VEL
LIN {X 0,Y 580.104,Z 515.601,A -85,B 0,C 180,E1 -1645.473,E2 -1645.473} C_VEL
LIN {X 0,Y 580.119,Z 520.78,A -85,B 0,C 180,E1 -1646.631,E2 -1646.631} C_VEL
LIN {X 0,Y 580.076,Z 524.668,A -85,B 0,C 180,E1 -1647.816,E2 -1647.816} C_VEL
LIN {X 0,Y 580.072,Z 527.685,A -85,B 0,C 180,E1 -1649.268,E2 -1649.268} C_VEL
LIN {X 0,Y 580.064,Z 528.92,A -85,B 0,C 180,E1 -1650.657,E2 -1650.657} C_VEL
LIN {X 0,Y 580.044,Z 528.616,A -85,B 0,C 180,E1 -1651.989,E2 -1651.989} C_VEL
LIN {X 0,Y 580.065,Z 526.941,A -85,B 0,C 180,E1 -1653.28,E2 -1653.28} C_VEL
LIN {X 0,Y 580.076,Z 523.934,A -85,B 0,C 180,E1 -1654.526,E2 -1654.526} C_VEL
LIN {X 0,Y 580.081,Z 519.677,A -85,B 0,C 180,E1 -1655.733,E2 -1655.733} C_VEL
LIN {X 0,Y 580.123,Z 514.108,A -85,B 0,C 180,E1 -1656.91,E2 -1656.91} C_VEL
LIN {X 0,Y 580.152,Z 507.106,A -85,B 0,C 180,E1 -1658.055,E2 -1658.055} C_VEL
LIN {X 0,Y 580.255,Z 498.4,A -85,B 0,C 180,E1 -1659.18,E2 -1659.18} C_VEL
LIN {X 0,Y 580.308,Z 489.525,A -85,B 0,C 180,E1 -1660.103,E2 -1660.103} C_VEL
LIN {X 0,Y 580.4,Z 479.337,A -85,B 0,C 180,E1 -1660.963,E2 -1660.963} C_VEL
LIN {X 0,Y 580.438,Z 468.706,A -85,B 0,C 180,E1 -1661.69,E2 -1661.69} C_VEL
LIN {X 0,Y 580.55,Z 456.818,A -85,B 0,C 180,E1 -1662.329,E2 -1662.329} C_VEL
LIN {X 0,Y 580.644,Z 445.074,A -85,B 0,C 180,E1 -1662.811,E2 -1662.811} C_VEL
LIN {X 0,Y 580.779,Z 432.099,A -85,B 0,C 180,E1 -1663.19,E2 -1663.19} C_VEL
LIN {X 0,Y 580.632,Z 427.063,A -85,B 0,C 180,E1 -1663.301,E2 -1663.301} C_VEL
LIN {X 0,Y 580.07,Z 423.465,A -85,B 0,C 180,E1 -1663.39,E2 -1663.39} C_VEL
LIN {X 0,Y 580.09,Z 417.811,A -85,B 0,C 180,E1 -1665.627,E2 -1665.627} C_VEL
LIN {X 0,Y 580.095,Z 411.342,A -85,B 0,C 180,E1 -1668.214,E2 -1668.214} C_VEL
LIN {X 0,Y 580.145,Z 404.587,A -85,B 0,C 180,E1 -1670.954,E2 -1670.954} C_VEL
LIN {X 0,Y 580.162,Z 398.202,A -85,B 0,C 180,E1 -1673.588,E2 -1673.588} C_VEL
LIN {X 0,Y 580.191,Z 392.139,A -85,B 0,C 180,E1 -1676.136,E2 -1676.136} C_VEL
LIN {X 0,Y 580.221,Z 386.116,A -85,B 0,C 180,E1 -1678.61,E2 -1678.61} C_VEL
LIN {X 0,Y 580.228,Z 380.267,A -85,B 0,C 180,E1 -1681.019,E2 -1681.019} C_VEL
LIN {X 0,Y 580.224,Z 373.81,A -85,B 0,C 180,E1 -1683.679,E2 -1683.679} C_VEL
LIN {X 0,Y 580.295,Z 368.203,A -85,B 0,C 180,E1 -1685.968,E2 -1685.968} C_VEL
LIN {X 0,Y 580.304,Z 368.204,A -85,B 0,C 180,E1 -1688.833,E2 -1688.833} C_VEL
LIN {X 0,Y 580.245,Z 368.207,A -85,B 0,C 180,E1 -1691.643,E2 -1691.643} C_VEL
LIN {X 0,Y 580.273,Z 368.205,A -85,B 0,C 180,E1 -1693.824,E2 -1693.824} C_VEL
LIN {X 0,Y 580.33,Z 368.195,A -85,B 0,C 180,E1 -1695.982,E2 -1695.982} C_VEL
LIN {X 0,Y 580.307,Z 368.198,A -85,B 0,C 180,E1 -1698.826,E2 -1698.826} C_VEL
LIN {X 0,Y 580.329,Z 368.198,A -85,B 0,C 180,E1 -1701.643,E2 -1701.643} C_VEL
LIN {X 0,Y 580.32,Z 368.201,A -85,B 0,C 180,E1 -1704.439,E2 -1704.439} C_VEL
LIN {X 0,Y 580.341,Z 368.197,A -85,B 0,C 180,E1 -1707.916,E2 -1707.916} C_VEL
LIN {X 0,Y 580.357,Z 368.361,A -85,B 0,C 180,E1 -1710.606,E2 -1710.606} C_VEL
LIN {X 0,Y 580.312,Z 372.946,A -85,B 0,C 180,E1 -1712.775,E2 -1712.775} C_VEL
LIN {X 0,Y 580.273,Z 378.866,A -85,B 0,C 180,E1 -1715.559,E2 -1715.559} C_VEL
LIN {X 0,Y 580.206,Z 384.894,A -85,B 0,C 180,E1 -1718.356,E2 -1718.356} C_VEL
LIN {X 0,Y 580.177,Z 391.143,A -85,B 0,C 180,E1 -1721.174,E2 -1721.174} C_VEL
LIN {X 0,Y 580.157,Z 398.18,A -85,B 0,C 180,E1 -1724.277,E2 -1724.277} C_VEL
LIN {X 0,Y 580.106,Z 404.234,A -85,B 0,C 180,E1 -1726.901,E2 -1726.901} C_VEL
LIN {X 0,Y 580.062,Z 411.081,A -85,B 0,C 180,E1 -1729.829,E2 -1729.829} C_VEL
LIN {X 0,Y 580.078,Z 418.133,A -85,B 0,C 180,E1 -1732.809,E2 -1732.809} C_VEL
LIN {X 0,Y 580.084,Z 419.474,A -85,B 0,C 180,E1 -1733.332,E2 -1733.332} C_VEL
LIN {X 0,Y 580.512,Z 425.809,A -85,B 0,C 180,E1 -1733.499,E2 -1733.499} C_VEL
LIN {X 0,Y 580.4,Z 435.873,A -85,B 0,C 180,E1 -1733.835,E2 -1733.835} C_VEL
LIN {X 0,Y 580.322,Z 447.442,A -85,B 0,C 180,E1 -1734.377,E2 -1734.377} C_VEL
LIN {X 0,Y 580.254,Z 456.876,A -85,B 0,C 180,E1 -1734.972,E2 -1734.972} C_VEL
LIN {X 0,Y 580.243,Z 465.519,A -85,B 0,C 180,E1 -1735.656,E2 -1735.656} C_VEL
LIN {X 0,Y 580.191,Z 473.405,A -85,B 0,C 180,E1 -1736.437,E2 -1736.437} C_VEL
LIN {X 0,Y 580.158,Z 479.714,A -85,B 0,C 180,E1 -1737.211,E2 -1737.211} C_VEL
LIN {X 0,Y 580.122,Z 486.082,A -85,B 0,C 180,E1 -1738.192,E2 -1738.192} C_VEL
LIN {X 0,Y 580.103,Z 490.125,A -85,B 0,C 180,E1 -1738.984,E2 -1738.984} C_VEL
LIN {X 0,Y 580.07,Z 494.676,A -85,B 0,C 180,E1 -1740.183,E2 -1740.183} C_VEL
LIN {X 0,Y 580.036,Z 497.566,A -85,B 0,C 180,E1 -1741.397,E2 -1741.397} C_VEL
LIN {X 0,Y 580.034,Z 498.637,A -85,B 0,C 180,E1 -1742.214,E2 -1742.214} C_VEL
LIN {X 0,Y 580.052,Z 498.92,A -85,B 0,C 180,E1 -1743.279,E2 -1743.279} C_VEL
LIN {X 0,Y 580.041,Z 498.64,A -85,B 0,C 180,E1 -1743.87,E2 -1743.87} C_VEL
LIN {X 0,Y 580.037,Z 497.54,A -85,B 0,C 180,E1 -1744.711,E2 -1744.711} C_VEL
LIN {X 0,Y 580.05,Z 495.233,A -85,B 0,C 180,E1 -1745.73,E2 -1745.73} C_VEL
LIN {X 0,Y 580.099,Z 490.986,A -85,B 0,C 180,E1 -1746.908,E2 -1746.908} C_VEL
LIN {X 0,Y 580.132,Z 485.181,A -85,B 0,C 180,E1 -1748.053,E2 -1748.053} C_VEL
LIN {X 0,Y 580.163,Z 478.525,A -85,B 0,C 180,E1 -1749.041,E2 -1749.041} C_VEL
LIN {X 0,Y 580.2,Z 470.719,A -85,B 0,C 180,E1 -1749.937,E2 -1749.937} C_VEL
LIN {X 0,Y 580.219,Z 461.592,A -85,B 0,C 180,E1 -1750.768,E2 -1750.768} C_VEL
LIN {X 0,Y 580.317,Z 451.866,A -85,B 0,C 180,E1 -1751.45,E2 -1751.45} C_VEL
LIN {X 0,Y 580.396,Z 443.197,A -85,B 0,C 180,E1 -1751.93,E2 -1751.93} C_VEL
LIN {X 0,Y 580.441,Z 433.83,A -85,B 0,C 180,E1 -1752.332,E2 -1752.332} C_VEL
LIN {X 0,Y 580.493,Z 424.033,A -85,B 0,C 180,E1 -1752.639,E2 -1752.639} C_VEL
LIN {X 0,Y 580.073,Z 419.349,A -85,B 0,C 180,E1 -1752.77,E2 -1752.77} C_VEL
LIN {X 0,Y 580.097,Z 412.583,A -85,B 0,C 180,E1 -1755.623,E2 -1755.623} C_VEL
LIN {X 0,Y 580.068,Z 406.508,A -85,B 0,C 180,E1 -1758.213,E2 -1758.213} C_VEL
LIN {X 0,Y 580.094,Z 400.162,A -85,B 0,C 180,E1 -1760.951,E2 -1760.951} C_VEL
LIN {X 0,Y 580.109,Z 394.149,A -85,B 0,C 180,E1 -1763.585,E2 -1763.585} C_VEL
LIN {X 0,Y 580.159,Z 388.422,A -85,B 0,C 180,E1 -1766.135,E2 -1766.135} C_VEL
LIN {X 0,Y 580.164,Z 383.047,A -85,B 0,C 180,E1 -1768.608,E2 -1768.608} C_VEL
LIN {X 0,Y 580.249,Z 377.951,A -85,B 0,C 180,E1 -1771.022,E2 -1771.022} C_VEL
LIN {X 0,Y 580.283,Z 371.175,A -85,B 0,C 180,E1 -1774.151,E2 -1774.151} C_VEL
LIN {X 0,Y 580.312,Z 368.201,A -85,B 0,C 180,E1 -1775.58,E2 -1775.58} C_VEL
LIN {X 0,Y 580.273,Z 368.208,A -85,B 0,C 180,E1 -1777.948,E2 -1777.948} C_VEL
LIN {X 0,Y 580.312,Z 368.201,A -85,B 0,C 180,E1 -1780.914,E2 -1780.914} C_VEL
LIN {X 0,Y 580.263,Z 368.206,A -85,B 0,C 180,E1 -1783.825,E2 -1783.825} C_VEL
LIN {X 0,Y 580.322,Z 368.202,A -85,B 0,C 180,E1 -1785.983,E2 -1785.983} C_VEL
LIN {X 0,Y 580.364,Z 368.195,A -85,B 0,C 180,E1 -1788.828,E2 -1788.828} C_VEL
LIN {X 0,Y 580.314,Z 368.2,A -85,B 0,C 180,E1 -1791.644,E2 -1791.644} C_VEL
LIN {X 0,Y 580.32,Z 368.198,A -85,B 0,C 180,E1 -1794.44,E2 -1794.44} C_VEL
LIN {X 0,Y 580.33,Z 368.197,A -85,B 0,C 180,E1 -1797.224,E2 -1797.224} C_VEL
LIN {X 0,Y 580.325,Z 368.197,A -85,B 0,C 180,E1 -1800,E2 -1800} C_VEL
LIN {X 0,Y 580.328,Z 368.197,A -85,B 0,C 180,E1 -1802.777,E2 -1802.777} C_VEL
LIN {X 0,Y 580.322,Z 368.198,A -85,B 0,C 180,E1 -1805.56,E2 -1805.56} C_VEL
LIN {X 0,Y 580.315,Z 368.2,A -85,B 0,C 180,E1 -1808.357,E2 -1808.357} C_VEL
LIN {X 0,Y 580.358,Z 368.197,A -85,B 0,C 180,E1 -1811.234,E2 -1811.234} C_VEL
LIN {X 0,Y 580.31,Z 368.2,A -85,B 0,C 180,E1 -1814.348,E2 -1814.348} C_VEL
LIN {X 0,Y 580.32,Z 368.2,A -85,B 0,C 180,E1 -1816.926,E2 -1816.926} C_VEL
LIN {X 0,Y 580.289,Z 368.202,A -85,B 0,C 180,E1 -1819.823,E2 -1819.823} C_VEL
LIN {X 0,Y 580.31,Z 368.199,A -85,B 0,C 180,E1 -1822.802,E2 -1822.802} C_VEL
LIN {X 0,Y 580.286,Z 368.203,A -85,B 0,C 180,E1 -1825.081,E2 -1825.081} C_VEL
LIN {X 0,Y 580.299,Z 368.2,A -85,B 0,C 180,E1 -1827.865,E2 -1827.865} C_VEL
LIN {X 0,Y 580.283,Z 368.202,A -85,B 0,C 180,E1 -1830.7,E2 -1830.7} C_VEL
LIN {X 0,Y 580.286,Z 368.202,A -85,B 0,C 180,E1 -1833.319,E2 -1833.319} C_VEL
LIN {X 0,Y 580.31,Z 368.2,A -85,B 0,C 180,E1 -1835.77,E2 -1835.77} C_VEL
LIN {X 0,Y 580.275,Z 368.207,A -85,B 0,C 180,E1 -1838.148,E2 -1838.148} C_VEL
LIN {X 0,Y 580.288,Z 368.205,A -85,B 0,C 180,E1 -1840.845,E2 -1840.845} C_VEL
LIN {X 0,Y 580.276,Z 368.205,A -85,B 0,C 180,E1 -1843.658,E2 -1843.658} C_VEL
LIN {X 0,Y 580.273,Z 368.204,A -85,B 0,C 180,E1 -1846.61,E2 -1846.61} C_VEL
LIN {X 0,Y 580.289,Z 368.203,A -85,B 0,C 180,E1 -1849.159,E2 -1849.159} C_VEL
LIN {X 0,Y 580.28,Z 368.203,A -85,B 0,C 180,E1 -1851.929,E2 -1851.929} C_VEL
LIN {X 0,Y 580.299,Z 368.202,A -85,B 0,C 180,E1 -1854.459,E2 -1854.459} C_VEL
LIN {X 0,Y 580.282,Z 368.206,A -85,B 0,C 180,E1 -1856.977,E2 -1856.977} C_VEL
LIN {X 0,Y 580.343,Z 368.366,A -85,B 0,C 180,E1 -1859.371,E2 -1859.371} C_VEL
LIN {X 0,Y 580.844,Z 371.929,A -85,B 0,C 180,E1 -1860.261,E2 -1860.261} C_VEL
LIN {X 0,Y 580.721,Z 381.898,A -85,B 0,C 180,E1 -1862.623,E2 -1862.623} C_VEL
LIN {X 0,Y 580.604,Z 394.225,A -85,B 0,C 180,E1 -1865.455,E2 -1865.455} C_VEL
LIN {X 0,Y 580.473,Z 407.081,A -85,B 0,C 180,E1 -1868.331,E2 -1868.331} C_VEL
LIN {X 0,Y 580.4,Z 418.857,A -85,B 0,C 180,E1 -1870.919,E2 -1870.919} C_VEL
LIN {X 0,Y 580.301,Z 432.315,A -85,B 0,C 180,E1 -1873.828,E2 -1873.828} C_VEL
LIN {X 0,Y 580.226,Z 445.774,A -85,B 0,C 180,E1 -1876.697,E2 -1876.697} C_VEL
LIN {X 0,Y 580.208,Z 450.137,A -85,B 0,C 180,E1 -1877.619,E2 -1877.619} C_VEL
LIN {X 0,Y 580.792,Z 455.042,A -85,B 0,C 180,E1 -1877.71,E2 -1877.71} C_VEL
LIN {X 0,Y 580.753,Z 468.278,A -85,B 0,C 180,E1 -1878.019,E2 -1878.019} C_VEL
LIN {X 0,Y 580.627,Z 480.416,A -85,B 0,C 180,E1 -1878.437,E2 -1878.437} C_VEL
LIN {X 0,Y 580.519,Z 492.664,A -85,B 0,C 180,E1 -1879.01,E2 -1879.01} C_VEL
LIN {X 0,Y 580.461,Z 504.229,A -85,B 0,C 180,E1 -1879.714,E2 -1879.714} C_VEL
LIN {X 0,Y 580.346,Z 514.62,A -85,B 0,C 180,E1 -1880.505,E2 -1880.505} C_VEL
LIN {X 0,Y 580.271,Z 523.13,A -85,B 0,C 180,E1 -1881.294,E2 -1881.294} C_VEL
LIN {X 0,Y 580.22,Z 530.975,A -85,B 0,C 180,E1 -1882.17,E2 -1882.17} C_VEL
LIN {X 0,Y 580.15,Z 538.683,A -85,B 0,C 180,E1 -1883.227,E2 -1883.227} C_VEL
LIN {X 0,Y 580.139,Z 545.689,A -85,B 0,C 180,E1 -1884.44,E2 -1884.44} C_VEL
LIN {X 0,Y 580.108,Z 550.378,A -85,B 0,C 180,E1 -1885.485,E2 -1885.485} C_VEL
LIN {X 0,Y 580.122,Z 553.963,A -85,B 0,C 180,E1 -1886.529,E2 -1886.529} C_VEL
LIN {X 0,Y 580.043,Z 555.814,A -85,B 0,C 180,E1 -1887.224,E2 -1887.224} C_VEL
LIN {X 0,Y 580.04,Z 557.203,A -85,B 0,C 180,E1 -1887.918,E2 -1887.918} C_VEL
LIN {X 0,Y 580.04,Z 558.786,A -85,B 0,C 180,E1 -1889.307,E2 -1889.307} C_VEL
LIN {X 0,Y 580.037,Z 559,A -85,B 0,C 180,E1 -1890.002,E2 -1890.002} C_VEL
LIN {X 0,Y 580.046,Z 558.183,A -85,B 0,C 180,E1 -1891.39,E2 -1891.39} C_VEL
LIN {X 0,Y 580.04,Z 557.197,A -85,B 0,C 180,E1 -1892.085,E2 -1892.085} C_VEL
LIN {X 0,Y 580.043,Z 555.805,A -85,B 0,C 180,E1 -1892.779,E2 -1892.779} C_VEL
LIN {X 0,Y 580.11,Z 552.891,A -85,B 0,C 180,E1 -1893.822,E2 -1893.822} C_VEL
LIN {X 0,Y 580.053,Z 548.944,A -85,B 0,C 180,E1 -1894.867,E2 -1894.867} C_VEL
LIN {X 0,Y 580.139,Z 542.869,A -85,B 0,C 180,E1 -1896.086,E2 -1896.086} C_VEL
LIN {X 0,Y 580.186,Z 536.227,A -85,B 0,C 180,E1 -1897.134,E2 -1897.134} C_VEL
LIN {X 0,Y 580.251,Z 527.979,A -85,B 0,C 180,E1 -1898.183,E2 -1898.183} C_VEL
LIN {X 0,Y 580.309,Z 519.523,A -85,B 0,C 180,E1 -1899.06,E2 -1899.06} C_VEL
LIN {X 0,Y 580.424,Z 509.079,A -85,B 0,C 180,E1 -1899.937,E2 -1899.937} C_VEL
LIN {X 0,Y 580.502,Z 498.735,A -85,B 0,C 180,E1 -1900.641,E2 -1900.641} C_VEL
LIN {X 0,Y 580.566,Z 487.566,A -85,B 0,C 180,E1 -1901.249,E2 -1901.249} C_VEL
LIN {X 0,Y 580.665,Z 475.734,A -85,B 0,C 180,E1 -1901.742,E2 -1901.742} C_VEL
LIN {X 0,Y 580.757,Z 462.301,A -85,B 0,C 180,E1 -1902.139,E2 -1902.139} C_VEL
LIN {X 0,Y 580.628,Z 452.878,A -85,B 0,C 180,E1 -1902.329,E2 -1902.329} C_VEL
LIN {X 0,Y 580.201,Z 450.07,A -85,B 0,C 180,E1 -1902.395,E2 -1902.395} C_VEL
LIN {X 0,Y 580.263,Z 437.347,A -85,B 0,C 180,E1 -1905.095,E2 -1905.095} C_VEL
LIN {X 0,Y 580.372,Z 423.889,A -85,B 0,C 180,E1 -1907.988,E2 -1907.988} C_VEL
LIN {X 0,Y 580.418,Z 410.655,A -85,B 0,C 180,E1 -1910.88,E2 -1910.88} C_VEL
LIN {X 0,Y 580.556,Z 398.655,A -85,B 0,C 180,E1 -1913.547,E2 -1913.547} C_VEL
LIN {X 0,Y 580.689,Z 386.021,A -85,B 0,C 180,E1 -1916.412,E2 -1916.412} C_VEL
LIN {X 0,Y 580.747,Z 375.07,A -85,B 0,C 180,E1 -1918.952,E2 -1918.952} C_VEL
LIN {X 0,Y 580.658,Z 370.169,A -85,B 0,C 180,E1 -1920.153,E2 -1920.153} C_VEL
LIN {X 0,Y 580.277,Z 368.207,A -85,B 0,C 180,E1 -1920.693,E2 -1920.693} C_VEL
LIN {X 0,Y 580.308,Z 368.199,A -85,B 0,C 180,E1 -1923.316,E2 -1923.316} C_VEL
LIN {X 0,Y 580.252,Z 368.204,A -85,B 0,C 180,E1 -1925.757,E2 -1925.757} C_VEL
LIN {X 0,Y 580.29,Z 368.206,A -85,B 0,C 180,E1 -1928.147,E2 -1928.147} C_VEL
LIN {X 0,Y 580.284,Z 368.199,A -85,B 0,C 180,E1 -1930.846,E2 -1930.846} C_VEL
LIN {X 0,Y 580.229,Z 368.213,A -85,B 0,C 180,E1 -1933.663,E2 -1933.663} C_VEL
LIN {X 0,Y 580.239,Z 368.205,A -85,B 0,C 180,E1 -1936.614,E2 -1936.614} C_VEL
LIN {X 0,Y 580.299,Z 368.202,A -85,B 0,C 180,E1 -1939.156,E2 -1939.156} C_VEL
LIN {X 0,Y 580.291,Z 368.198,A -85,B 0,C 180,E1 -1941.928,E2 -1941.928} C_VEL
LIN {X 0,Y 580.257,Z 368.208,A -85,B 0,C 180,E1 -1944.453,E2 -1944.453} C_VEL
LIN {X 0,Y 580.293,Z 368.197,A -85,B 0,C 180,E1 -1946.975,E2 -1946.975} C_VEL
LIN {X 0,Y 580.287,Z 368.202,A -85,B 0,C 180,E1 -1949.424,E2 -1949.424} C_VEL
LIN {X 0,Y 580.25,Z 368.203,A -85,B 0,C 180,E1 -1952.151,E2 -1952.151} C_VEL
LIN {X 0,Y 580.237,Z 368.21,A -85,B 0,C 180,E1 -1954.917,E2 -1954.917} C_VEL
LIN {X 0,Y 580.289,Z 368.202,A -85,B 0,C 180,E1 -1957.197,E2 -1957.197} C_VEL
LIN {X 0,Y 580.273,Z 368.2,A -85,B 0,C 180,E1 -1959.437,E2 -1959.437} C_VEL
LIN {X 0,Y 580.267,Z 368.202,A -85,B 0,C 180,E1 -1961.645,E2 -1961.645} C_VEL
LIN {X 0,Y 580.278,Z 368.205,A -85,B 0,C 180,E1 -1963.825,E2 -1963.825} C_VEL
LIN {X 0,Y 580.325,Z 368.2,A -85,B 0,C 180,E1 -1965.983,E2 -1965.983} C_VEL
LIN {X 0,Y 580.309,Z 368.197,A -85,B 0,C 180,E1 -1968.827,E2 -1968.827} C_VEL
LIN {X 0,Y 580.284,Z 368.201,A -85,B 0,C 180,E1 -1971.643,E2 -1971.643} C_VEL
LIN {X 0,Y 580.307,Z 368.199,A -85,B 0,C 180,E1 -1974.44,E2 -1974.44} C_VEL
LIN {X 0,Y 580.184,Z 368.266,A -85,B 0,C 180,E1 -1976.701,E2 -1976.701} C_VEL
LIN {X 0,Y 580.222,Z 375.321,A -85,B 0,C 180,E1 -1979.306,E2 -1979.306} C_VEL
LIN {X 0,Y 580.242,Z 380.799,A -85,B 0,C 180,E1 -1981.388,E2 -1981.388} C_VEL
LIN {X 0,Y 580.23,Z 387.744,A -85,B 0,C 180,E1 -1984.167,E2 -1984.167} C_VEL
LIN {X 0,Y 580.214,Z 393.806,A -85,B 0,C 180,E1 -1986.661,E2 -1986.661} C_VEL
LIN {X 0,Y 580.19,Z 399.541,A -85,B 0,C 180,E1 -1989.06,E2 -1989.06} C_VEL
LIN {X 0,Y 580.153,Z 406.418,A -85,B 0,C 180,E1 -1991.884,E2 -1991.884} C_VEL
LIN {X 0,Y 580.12,Z 413.487,A -85,B 0,C 180,E1 -1994.738,E2 -1994.738} C_VEL
LIN {X 0,Y 580.054,Z 420.761,A -85,B 0,C 180,E1 -1997.632,E2 -1997.632} C_VEL
LIN {X 0,Y 580.094,Z 423.474,A -85,B 0,C 180,E1 -1998.704,E2 -1998.704} C_VEL
LIN {X 0,Y 580.809,Z 429.431,A -85,B 0,C 180,E1 -1998.84,E2 -1998.84} C_VEL
LIN {X 0,Y 580.709,Z 441.422,A -85,B 0,C 180,E1 -1999.158,E2 -1999.158} C_VEL
LIN {X 0,Y 580.648,Z 447.855,A -85,B 0,C 180,E1 -1999.382,E2 -1999.382} C_VEL
LIN {X 0,Y 580.019,Z 453.36,A -85,B 0,C 180,E1 -1999.592,E2 -1999.592} C_VEL
LIN {X 0,Y 577.136,Z 462.135,A -85,B 0,C 180,E1 -1999.962,E2 -1999.962} C_VEL
LIN {X 0,Y 574.175,Z 470.548,A -85,B 0,C 180,E1 -2000.399,E2 -2000.399} C_VEL
LIN {X 0,Y 573.412,Z 475.368,A -85,B 0,C 180,E1 -2000.713,E2 -2000.713} C_VEL
LIN {X 0,Y 573.332,Z 486.283,A -85,B 0,C 180,E1 -2001.576,E2 -2001.576} C_VEL
LIN {X 0,Y 573.186,Z 495.915,A -85,B 0,C 180,E1 -2002.53,E2 -2002.53} C_VEL
LIN {X 0,Y 573.13,Z 503.773,A -85,B 0,C 180,E1 -2003.486,E2 -2003.486} C_VEL
LIN {X 0,Y 573.054,Z 510.307,A -85,B 0,C 180,E1 -2004.451,E2 -2004.451} C_VEL
LIN {X 0,Y 573.025,Z 515.68,A -85,B 0,C 180,E1 -2005.421,E2 -2005.421} C_VEL
LIN {X 0,Y 573.028,Z 520.292,A -85,B 0,C 180,E1 -2006.45,E2 -2006.45} C_VEL
LIN {X 0,Y 572.979,Z 524.68,A -85,B 0,C 180,E1 -2007.781,E2 -2007.781} C_VEL
LIN {X 0,Y 572.944,Z 526.52,A -85,B 0,C 180,E1 -2008.58,E2 -2008.58} C_VEL
LIN {X 0,Y 572.974,Z 527.926,A -85,B 0,C 180,E1 -2009.439,E2 -2009.439} C_VEL
LIN {X 0,Y 572.945,Z 528.687,A -85,B 0,C 180,E1 -2010.193,E2 -2010.193} C_VEL
LIN {X 0,Y 572.959,Z 528.997,A -85,B 0,C 180,E1 -2011.009,E2 -2011.009} C_VEL
LIN {X 0,Y 572.955,Z 528.482,A -85,B 0,C 180,E1 -2012.18,E2 -2012.18} C_VEL
LIN {X 0,Y 572.969,Z 526.547,A -85,B 0,C 180,E1 -2013.502,E2 -2013.502} C_VEL
LIN {X 0,Y 572.993,Z 523.435,A -85,B 0,C 180,E1 -2014.736,E2 -2014.736} C_VEL
LIN {X 0,Y 573.016,Z 518.536,A -85,B 0,C 180,E1 -2016.066,E2 -2016.066} C_VEL
LIN {X 0,Y 573.046,Z 513.26,A -85,B 0,C 180,E1 -2017.138,E2 -2017.138} C_VEL
LIN {X 0,Y 573.114,Z 506.042,A -85,B 0,C 180,E1 -2018.295,E2 -2018.295} C_VEL
LIN {X 0,Y 573.21,Z 498.324,A -85,B 0,C 180,E1 -2019.289,E2 -2019.289} C_VEL
LIN {X 0,Y 573.285,Z 488.713,A -85,B 0,C 180,E1 -2020.291,E2 -2020.291} C_VEL
LIN {X 0,Y 573.393,Z 477.742,A -85,B 0,C 180,E1 -2021.208,E2 -2021.208} C_VEL
LIN {X 0,Y 573.452,Z 466.376,A -85,B 0,C 180,E1 -2021.961,E2 -2021.961} C_VEL
LIN {X 0,Y 573.593,Z 455.633,A -85,B 0,C 180,E1 -2022.523,E2 -2022.523} C_VEL
LIN {X 0,Y 573.734,Z 443.786,A -85,B 0,C 180,E1 -2023,E2 -2023} C_VEL
LIN {X 0,Y 573.847,Z 430.704,A -85,B 0,C 180,E1 -2023.371,E2 -2023.371} C_VEL
LIN {X 0,Y 573.296,Z 425.517,A -85,B 0,C 180,E1 -2023.49,E2 -2023.49} C_VEL
LIN {X 0,Y 572.984,Z 423.49,A -85,B 0,C 180,E1 -2023.536,E2 -2023.536} C_VEL
LIN {X 0,Y 572.997,Z 416.459,A -85,B 0,C 180,E1 -2026.357,E2 -2026.357} C_VEL
LIN {X 0,Y 573.042,Z 408.737,A -85,B 0,C 180,E1 -2029.498,E2 -2029.498} C_VEL
LIN {X 0,Y 573.057,Z 402.263,A -85,B 0,C 180,E1 -2032.178,E2 -2032.178} C_VEL
LIN {X 0,Y 573.133,Z 394.99,A -85,B 0,C 180,E1 -2035.243,E2 -2035.243} C_VEL
LIN {X 0,Y 573.152,Z 388.834,A -85,B 0,C 180,E1 -2037.787,E2 -2037.787} C_VEL
LIN {X 0,Y 573.134,Z 381.926,A -85,B 0,C 180,E1 -2040.626,E2 -2040.626} C_VEL
LIN {X 0,Y 573.156,Z 376.22,A -85,B 0,C 180,E1 -2043.018,E2 -2043.018} C_VEL
LIN {X 0,Y 573.264,Z 369.08,A -85,B 0,C 180,E1 -2045.943,E2 -2045.943} C_VEL
LIN {X 0,Y 573.254,Z 369.08,A -85,B 0,C 180,E1 -2048.708,E2 -2048.708} C_VEL
LIN {X 0,Y 573.203,Z 369.083,A -85,B 0,C 180,E1 -2051.409,E2 -2051.409} C_VEL
LIN {X 0,Y 573.246,Z 369.083,A -85,B 0,C 180,E1 -2053.62,E2 -2053.62} C_VEL
LIN {X 0,Y 573.276,Z 369.074,A -85,B 0,C 180,E1 -2055.806,E2 -2055.806} C_VEL
LIN {X 0,Y 573.265,Z 369.076,A -85,B 0,C 180,E1 -2058.744,E2 -2058.744} C_VEL
LIN {X 0,Y 573.284,Z 369.077,A -85,B 0,C 180,E1 -2061.539,E2 -2061.539} C_VEL
LIN {X 0,Y 573.287,Z 369.077,A -85,B 0,C 180,E1 -2064.37,E2 -2064.37} C_VEL
LIN {X 0,Y 573.31,Z 369.073,A -85,B 0,C 180,E1 -2067.891,E2 -2067.891} C_VEL
LIN {X 0,Y 573.322,Z 369.113,A -85,B 0,C 180,E1 -2070.525,E2 -2070.525} C_VEL
LIN {X 0,Y 573.253,Z 373.874,A -85,B 0,C 180,E1 -2072.809,E2 -2072.809} C_VEL
